LIN {X 0,Y 239.846,Z 548.939,A -85,B 0,C 180,E1 -19168.321,E2 -19168.321} C_VEL
LIN {X 0,Y 239.916,Z 549.699,A -85,B 0,C 180,E1 -19170,E2 -19170} C_VEL
LIN {X 0,Y 239.751,Z 550.198,A -85,B 0,C 180,E1 -19173.361,E2 -19173.361} C_VEL
LIN {X 0,Y 239.899,Z 549.378,A -85,B 0,C 180,E1 -19176.729,E2 -19176.729} C_VEL
LIN {X 0,Y 240.489,Z 547.237,A -85,B 0,C 180,E1 -19180.098,E2 -19180.098} C_VEL
LIN {X 0,Y 241.611,Z 543.73,A -85,B 0,C 180,E1 -19183.456,E2 -19183.456} C_VEL
LIN {X 0,Y 243.585,Z 538.761,A -85,B 0,C 180,E1 -19186.769,E2 -19186.769} C_VEL
LIN {X 0,Y 245.464,Z 533.916,A -85,B 0,C 180,E1 -19189.262,E2 -19189.262} C_VEL
LIN {X 0,Y 248.227,Z 527.144,A -85,B 0,C 180,E1 -19192.033,E2 -19192.033} C_VEL
LIN {X 0,Y 251.636,Z 518.678,A -85,B 0,C 180,E1 -19194.767,E2 -19194.767} C_VEL
LIN {X 0,Y 255.078,Z 509.872,A -85,B 0,C 180,E1 -19197.039,E2 -19197.039} C_VEL
LIN {X 0,Y 258.85,Z 499.246,A -85,B 0,C 180,E1 -19199.255,E2 -19199.255} C_VEL
LIN {X 0,Y 262.242,Z 488.539,A -85,B 0,C 180,E1 -19201.056,E2 -19201.056} C_VEL
LIN {X 0,Y 265.684,Z 476.851,A -85,B 0,C 180,E1 -19202.612,E2 -19202.612} C_VEL
LIN {X 0,Y 268.817,Z 464.011,A -85,B 0,C 180,E1 -19203.974,E2 -19203.974} C_VEL
LIN {X 0,Y 271.609,Z 450.631,A -85,B 0,C 180,E1 -19205.036,E2 -19205.036} C_VEL
LIN {X 0,Y 273.793,Z 436.72,A -85,B 0,C 180,E1 -19205.842,E2 -19205.842} C_VEL
LIN {X 0,Y 275.284,Z 422.47,A -85,B 0,C 180,E1 -19206.395,E2 -19206.395} C_VEL
LIN {X 0,Y 279.07,Z 347.973,A -85,B 0,C 180,E1 -19208.307,E2 -19208.307} C_VEL
LIN {X 0,Y 278.474,Z 345.19,A -85,B 0,C 180,E1 -19208.52,E2 -19208.52} C_VEL
LIN {X 0,Y 272.199,Z 331.36,A -85,B 0,C 180,E1 -19210.309,E2 -19210.309} C_VEL
LIN {X 0,Y 266.418,Z 320.049,A -85,B 0,C 180,E1 -19212.032,E2 -19212.032} C_VEL
LIN {X 0,Y 260.658,Z 310.039,A -85,B 0,C 180,E1 -19213.842,E2 -19213.842} C_VEL
LIN {X 0,Y 255.666,Z 301.72,A -85,B 0,C 180,E1 -19215.523,E2 -19215.523} C_VEL
LIN {X 0,Y 251.265,Z 295.251,A -85,B 0,C 180,E1 -19217.083,E2 -19217.083} C_VEL
LIN {X 0,Y 247.968,Z 290.346,A -85,B 0,C 180,E1 -19218.331,E2 -19218.331} C_VEL
LIN {X 0,Y 244.184,Z 284.789,A -85,B 0,C 180,E1 -19219.908,E2 -19219.908} C_VEL
LIN {X 0,Y 242.91,Z 280.592,A -85,B 0,C 180,E1 -19222.583,E2 -19222.583} C_VEL
LIN {X 0,Y 241.985,Z 277.932,A -85,B 0,C 180,E1 -19224.487,E2 -19224.487} C_VEL
LIN {X 0,Y 241.974,Z 277.96,A -85,B 0,C 180,E1 -19228.478,E2 -19228.478} C_VEL
LIN {X 0,Y 242.007,Z 277.954,A -85,B 0,C 180,E1 -19232.31,E2 -19232.31} C_VEL
LIN {X 0,Y 242.055,Z 277.948,A -85,B 0,C 180,E1 -19236.014,E2 -19236.014} C_VEL
LIN {X 0,Y 242.035,Z 277.95,A -85,B 0,C 180,E1 -19239.606,E2 -19239.606} C_VEL
LIN {X 0,Y 242.161,Z 277.935,A -85,B 0,C 180,E1 -19243.276,E2 -19243.276} C_VEL
LIN {X 0,Y 242.182,Z 277.929,A -85,B 0,C 180,E1 -19248.277,E2 -19248.277} C_VEL
LIN {X 0,Y 242.422,Z 277.903,A -85,B 0,C 180,E1 -19251.663,E2 -19251.663} C_VEL
LIN {X 0,Y 242.254,Z 277.935,A -85,B 0,C 180,E1 -19255.005,E2 -19255.005} C_VEL
LIN {X 0,Y 242.631,Z 277.881,A -85,B 0,C 180,E1 -19258.338,E2 -19258.338} C_VEL
LIN {X 0,Y 242.631,Z 277.874,A -85,B 0,C 180,E1 -19261.658,E2 -19261.658} C_VEL
LIN {X 0,Y 242.419,Z 277.905,A -85,B 0,C 180,E1 -19266.732,E2 -19266.732} C_VEL
LIN {X 0,Y 242.307,Z 277.915,A -85,B 0,C 180,E1 -19270.02,E2 -19270.02} C_VEL
LIN {X 0,Y 242.158,Z 277.944,A -85,B 0,C 180,E1 -19275.139,E2 -19275.139} C_VEL
LIN {X 0,Y 242.065,Z 277.955,A -85,B 0,C 180,E1 -19278.622,E2 -19278.622} C_VEL
LIN {X 0,Y 242.004,Z 277.965,A -85,B 0,C 180,E1 -19282.178,E2 -19282.178} C_VEL
LIN {X 0,Y 242.085,Z 277.957,A -85,B 0,C 180,E1 -19285.468,E2 -19285.468} C_VEL
LIN {X 0,Y 242.865,Z 280.47,A -85,B 0,C 180,E1 -19285.896,E2 -19285.896} C_VEL
LIN {X 0,Y 244.734,Z 282.697,A -85,B 0,C 180,E1 -19286.658,E2 -19286.658} C_VEL
LIN {X 0,Y 246.03,Z 283.589,A -85,B 0,C 180,E1 -19287.137,E2 -19287.137} C_VEL
LIN {X 0,Y 247.872,Z 286.714,A -85,B 0,C 180,E1 -19287.891,E2 -19287.891} C_VEL
LIN {X 0,Y 249.981,Z 289.004,A -85,B 0,C 180,E1 -19288.662,E2 -19288.662} C_VEL
LIN {X 0,Y 252.783,Z 292.768,A -85,B 0,C 180,E1 -19289.68,E2 -19289.68} C_VEL
LIN {X 0,Y 257.721,Z 299.629,A -85,B 0,C 180,E1 -19291.374,E2 -19291.374} C_VEL
LIN {X 0,Y 265.051,Z 311.16,A -85,B 0,C 180,E1 -19293.719,E2 -19293.719} C_VEL
LIN {X 0,Y 272.108,Z 323.656,A -85,B 0,C 180,E1 -19295.812,E2 -19295.812} C_VEL
LIN {X 0,Y 278.325,Z 336.16,A -85,B 0,C 180,E1 -19297.559,E2 -19297.559} C_VEL
LIN {X 0,Y 279.569,Z 338.86,A -85,B 0,C 180,E1 -19297.9,E2 -19297.9} C_VEL
LIN {X 0,Y 275.587,Z 413.281,A -85,B 0,C 180,E1 -19299.801,E2 -19299.801} C_VEL
LIN {X 0,Y 274.052,Z 427.455,A -85,B 0,C 180,E1 -19300.42,E2 -19300.42} C_VEL
LIN {X 0,Y 271.873,Z 441.305,A -85,B 0,C 180,E1 -19301.301,E2 -19301.301} C_VEL
LIN {X 0,Y 269.63,Z 452.971,A -85,B 0,C 180,E1 -19302.304,E2 -19302.304} C_VEL
LIN {X 0,Y 266.75,Z 465.144,A -85,B 0,C 180,E1 -19303.631,E2 -19303.631} C_VEL
LIN {X 0,Y 263.406,Z 477.1,A -85,B 0,C 180,E1 -19305.276,E2 -19305.276} C_VEL
LIN {X 0,Y 259.874,Z 488.093,A -85,B 0,C 180,E1 -19307.164,E2 -19307.164} C_VEL
LIN {X 0,Y 256.22,Z 498.314,A -85,B 0,C 180,E1 -19309.35,E2 -19309.35} C_VEL
LIN {X 0,Y 252.677,Z 507.464,A -85,B 0,C 180,E1 -19311.795,E2 -19311.795} C_VEL
LIN {X 0,Y 249.407,Z 515.53,A -85,B 0,C 180,E1 -19314.512,E2 -19314.512} C_VEL
LIN {X 0,Y 246.666,Z 521.907,A -85,B 0,C 180,E1 -19317.226,E2 -19317.226} C_VEL
LIN {X 0,Y 244.406,Z 527.11,A -85,B 0,C 180,E1 -19320.06,E2 -19320.06} C_VEL
LIN {X 0,Y 242.442,Z 531.556,A -85,B 0,C 180,E1 -19323.301,E2 -19323.301} C_VEL
LIN {X 0,Y 241.219,Z 534.09,A -85,B 0,C 180,E1 -19325.928,E2 -19325.928} C_VEL
LIN {X 0,Y 240.214,Z 536.197,A -85,B 0,C 180,E1 -19329.447,E2 -19329.447} C_VEL
LIN {X 0,Y 239.65,Z 536.862,A -85,B 0,C 180,E1 -19332.947,E2 -19332.947} C_VEL
LIN {X 0,Y 239.567,Z 536.099,A -85,B 0,C 180,E1 -19336.427,E2 -19336.427} C_VEL
LIN {X 0,Y 239.643,Z 533.956,A -85,B 0,C 180,E1 -19339.866,E2 -19339.866} C_VEL
LIN {X 0,Y 240.177,Z 530.391,A -85,B 0,C 180,E1 -19343.279,E2 -19343.279} C_VEL
LIN {X 0,Y 240.703,Z 526.769,A -85,B 0,C 180,E1 -19345.814,E2 -19345.814} C_VEL
LIN {X 0,Y 241.452,Z 522.2,A -85,B 0,C 180,E1 -19348.332,E2 -19348.332} C_VEL
LIN {X 0,Y 242.697,Z 515.61,A -85,B 0,C 180,E1 -19351.245,E2 -19351.245} C_VEL
LIN {X 0,Y 244.491,Z 507.418,A -85,B 0,C 180,E1 -19354.121,E2 -19354.121} C_VEL
LIN {X 0,Y 246.418,Z 498.852,A -85,B 0,C 180,E1 -19356.551,E2 -19356.551} C_VEL
LIN {X 0,Y 248.723,Z 488.467,A -85,B 0,C 180,E1 -19358.941,E2 -19358.941} C_VEL
LIN {X 0,Y 251.085,Z 477.181,A -85,B 0,C 180,E1 -19361.039,E2 -19361.039} C_VEL
LIN {X 0,Y 253.256,Z 465.291,A -85,B 0,C 180,E1 -19362.827,E2 -19362.827} C_VEL
LIN {X 0,Y 254.994,Z 454.356,A -85,B 0,C 180,E1 -19364.158,E2 -19364.158} C_VEL
LIN {X 0,Y 256.893,Z 440.565,A -85,B 0,C 180,E1 -19365.47,E2 -19365.47} C_VEL
LIN {X 0,Y 258.331,Z 426.742,A -85,B 0,C 180,E1 -19366.446,E2 -19366.446} C_VEL
LIN {X 0,Y 259.427,Z 412.336,A -85,B 0,C 180,E1 -19367.134,E2 -19367.134} C_VEL
LIN {X 0,Y 262.832,Z 324.192,A -85,B 0,C 180,E1 -19369.505,E2 -19369.505} C_VEL
LIN {X 0,Y 255.522,Z 305.251,A -85,B 0,C 180,E1 -19371.012,E2 -19371.012} C_VEL
LIN {X 0,Y 250.035,Z 293.105,A -85,B 0,C 180,E1 -19372.147,E2 -19372.147} C_VEL
LIN {X 0,Y 242.324,Z 279.276,A -85,B 0,C 180,E1 -19373.732,E2 -19373.732} C_VEL
LIN {X 0,Y 242.049,Z 277.961,A -85,B 0,C 180,E1 -19373.835,E2 -19373.835} C_VEL
LIN {X 0,Y 241.998,Z 277.966,A -85,B 0,C 180,E1 -19377.688,E2 -19377.688} C_VEL
LIN {X 0,Y 241.965,Z 277.968,A -85,B 0,C 180,E1 -19381.521,E2 -19381.521} C_VEL
LIN {X 0,Y 242.018,Z 277.961,A -85,B 0,C 180,E1 -19385.605,E2 -19385.605} C_VEL
LIN {X 0,Y 241.999,Z 277.956,A -85,B 0,C 180,E1 -19389.71,E2 -19389.71} C_VEL
LIN {X 0,Y 242,Z 277.963,A -85,B 0,C 180,E1 -19394.185,E2 -19394.185} C_VEL
LIN {X 0,Y 242.027,Z 277.954,A -85,B 0,C 180,E1 -19398.1,E2 -19398.1} C_VEL
LIN {X 0,Y 242.003,Z 277.958,A -85,B 0,C 180,E1 -19402.424,E2 -19402.424} C_VEL
LIN {X 0,Y 241.982,Z 277.959,A -85,B 0,C 180,E1 -19406.511,E2 -19406.511} C_VEL
LIN {X 0,Y 242.028,Z 277.956,A -85,B 0,C 180,E1 -19410.589,E2 -19410.589} C_VEL
LIN {X 0,Y 242.06,Z 277.941,A -85,B 0,C 180,E1 -19414.185,E2 -19414.185} C_VEL
LIN {X 0,Y 242.046,Z 277.959,A -85,B 0,C 180,E1 -19418.299,E2 -19418.299} C_VEL
LIN {X 0,Y 242.157,Z 277.945,A -85,B 0,C 180,E1 -19423.28,E2 -19423.28} C_VEL
LIN {X 0,Y 242.174,Z 277.943,A -85,B 0,C 180,E1 -19428.282,E2 -19428.282} C_VEL
LIN {X 0,Y 242.395,Z 277.902,A -85,B 0,C 180,E1 -19431.667,E2 -19431.667} C_VEL
LIN {X 0,Y 242.253,Z 277.923,A -85,B 0,C 180,E1 -19435.009,E2 -19435.009} C_VEL
LIN {X 0,Y 242.632,Z 277.888,A -85,B 0,C 180,E1 -19438.342,E2 -19438.342} C_VEL
LIN {X 0,Y 242.632,Z 277.873,A -85,B 0,C 180,E1 -19441.662,E2 -19441.662} C_VEL
LIN {X 0,Y 242.365,Z 277.899,A -85,B 0,C 180,E1 -19443.351,E2 -19443.351} C_VEL
LIN {X 0,Y 241.593,Z 278.005,A -85,B 0,C 180,E1 -19444.738,E2 -19444.738} C_VEL
LIN {X 0,Y 238.745,Z 278.37,A -85,B 0,C 180,E1 -19447.002,E2 -19447.002} C_VEL
LIN {X 0,Y 235.536,Z 278.767,A -85,B 0,C 180,E1 -19449.792,E2 -19449.792} C_VEL
LIN {X 0,Y 235.167,Z 278.802,A -85,B 0,C 180,E1 -19450.758,E2 -19450.758} C_VEL
LIN {X 0,Y 235.105,Z 278.82,A -85,B 0,C 180,E1 -19455.609,E2 -19455.609} C_VEL
LIN {X 0,Y 235.005,Z 278.83,A -85,B 0,C 180,E1 -19459.208,E2 -19459.208} C_VEL
LIN {X 0,Y 234.952,Z 278.839,A -85,B 0,C 180,E1 -19462.886,E2 -19462.886} C_VEL
LIN {X 0,Y 234.97,Z 278.838,A -85,B 0,C 180,E1 -19466.659,E2 -19466.659} C_VEL
LIN {X 0,Y 234.933,Z 278.842,A -85,B 0,C 180,E1 -19470.57,E2 -19470.57} C_VEL
LIN {X 0,Y 234.935,Z 278.843,A -85,B 0,C 180,E1 -19474.639,E2 -19474.639} C_VEL
LIN {X 0,Y 234.944,Z 278.845,A -85,B 0,C 180,E1 -19478.946,E2 -19478.946} C_VEL
LIN {X 0,Y 234.89,Z 278.85,A -85,B 0,C 180,E1 -19483.488,E2 -19483.488} C_VEL
LIN {X 0,Y 234.895,Z 278.874,A -85,B 0,C 180,E1 -19488.167,E2 -19488.167} C_VEL
LIN {X 0,Y 236.892,Z 286.452,A -85,B 0,C 180,E1 -19491.308,E2 -19491.308} C_VEL
LIN {X 0,Y 244.745,Z 303.391,A -85,B 0,C 180,E1 -19493.084,E2 -19493.084} C_VEL
LIN {X 0,Y 252.555,Z 322.958,A -85,B 0,C 180,E1 -19494.805,E2 -19494.805} C_VEL
LIN {X 0,Y 253.857,Z 327.02,A -85,B 0,C 180,E1 -19495.104,E2 -19495.104} C_VEL
LIN {X 0,Y 256.076,Z 343.908,A -85,B 0,C 180,E1 -19495.922,E2 -19495.922} C_VEL
LIN {X 0,Y 252.934,Z 424.435,A -85,B 0,C 180,E1 -19498.135,E2 -19498.135} C_VEL
LIN {X 0,Y 251.91,Z 437.762,A -85,B 0,C 180,E1 -19498.752,E2 -19498.752} C_VEL
LIN {X 0,Y 250.233,Z 451.111,A -85,B 0,C 180,E1 -19499.633,E2 -19499.633} C_VEL
LIN {X 0,Y 248.32,Z 463.814,A -85,B 0,C 180,E1 -19500.777,E2 -19500.777} C_VEL
LIN {X 0,Y 246.163,Z 476.754,A -85,B 0,C 180,E1 -19502.311,E2 -19502.311} C_VEL
LIN {X 0,Y 244.22,Z 486.606,A -85,B 0,C 180,E1 -19503.74,E2 -19503.74} C_VEL
LIN {X 0,Y 241.878,Z 497.961,A -85,B 0,C 180,E1 -19505.769,E2 -19505.769} C_VEL
LIN {X 0,Y 239.496,Z 508.241,A -85,B 0,C 180,E1 -19508.029,E2 -19508.029} C_VEL
LIN {X 0,Y 237.408,Z 517.546,A -85,B 0,C 180,E1 -19510.547,E2 -19510.547} C_VEL
LIN {X 0,Y 235.808,Z 525.288,A -85,B 0,C 180,E1 -19513.107,E2 -19513.107} C_VEL
LIN {X 0,Y 234.372,Z 532.651,A -85,B 0,C 180,E1 -19516.12,E2 -19516.12} C_VEL
LIN {X 0,Y 233.48,Z 537.791,A -85,B 0,C 180,E1 -19518.717,E2 -19518.717} C_VEL
LIN {X 0,Y 232.927,Z 543.07,A -85,B 0,C 180,E1 -19522.196,E2 -19522.196} C_VEL
LIN {X 0,Y 232.701,Z 546.505,A -85,B 0,C 180,E1 -19525.335,E2 -19525.335} C_VEL
LIN {X 0,Y 232.758,Z 548.66,A -85,B 0,C 180,E1 -19528.27,E2 -19528.27} C_VEL
LIN {X 0,Y 232.825,Z 549.454,A -85,B 0,C 180,E1 -19530,E2 -19530} C_VEL
LIN {X 0,Y 232.662,Z 550.012,A -85,B 0,C 180,E1 -19533.463,E2 -19533.463} C_VEL
LIN {X 0,Y 232.82,Z 549.246,A -85,B 0,C 180,E1 -19536.935,E2 -19536.935} C_VEL
LIN {X 0,Y 233.47,Z 547.162,A -85,B 0,C 180,E1 -19540.405,E2 -19540.405} C_VEL
LIN {X 0,Y 234.687,Z 543.715,A -85,B 0,C 180,E1 -19543.861,E2 -19543.861} C_VEL
LIN {X 0,Y 236.758,Z 538.813,A -85,B 0,C 180,E1 -19547.267,E2 -19547.267} C_VEL
LIN {X 0,Y 238.627,Z 534.303,A -85,B 0,C 180,E1 -19549.707,E2 -19549.707} C_VEL
LIN {X 0,Y 241.645,Z 527.347,A -85,B 0,C 180,E1 -19552.666,E2 -19552.666} C_VEL
LIN {X 0,Y 245.222,Z 518.966,A -85,B 0,C 180,E1 -19555.46,E2 -19555.46} C_VEL
LIN {X 0,Y 248.79,Z 510.258,A -85,B 0,C 180,E1 -19557.781,E2 -19557.781} C_VEL
LIN {X 0,Y 252.717,Z 499.747,A -85,B 0,C 180,E1 -19560.037,E2 -19560.037} C_VEL
LIN {X 0,Y 256.218,Z 489.183,A -85,B 0,C 180,E1 -19561.871,E2 -19561.871} C_VEL
LIN {X 0,Y 259.781,Z 477.673,A -85,B 0,C 180,E1 -19563.449,E2 -19563.449} C_VEL
LIN {X 0,Y 263.013,Z 465.076,A -85,B 0,C 180,E1 -19564.83,E2 -19564.83} C_VEL
LIN {X 0,Y 265.898,Z 452.049,A -85,B 0,C 180,E1 -19565.904,E2 -19565.904} C_VEL
LIN {X 0,Y 268.244,Z 438.06,A -85,B 0,C 180,E1 -19566.762,E2 -19566.762} C_VEL
LIN {X 0,Y 269.928,Z 423.494,A -85,B 0,C 180,E1 -19567.36,E2 -19567.36} C_VEL
LIN {X 0,Y 273.887,Z 349.141,A -85,B 0,C 180,E1 -19569.299,E2 -19569.299} C_VEL
LIN {X 0,Y 268.082,Z 336.015,A -85,B 0,C 180,E1 -19571.032,E2 -19571.032} C_VEL
LIN {X 0,Y 262.07,Z 324.165,A -85,B 0,C 180,E1 -19572.906,E2 -19572.906} C_VEL
LIN {X 0,Y 256.592,Z 314.442,A -85,B 0,C 180,E1 -19574.715,E2 -19574.715} C_VEL
LIN {X 0,Y 251.898,Z 306.619,A -85,B 0,C 180,E1 -19576.369,E2 -19576.369} C_VEL
LIN {X 0,Y 248.032,Z 300.769,A -85,B 0,C 180,E1 -19577.805,E2 -19577.805} C_VEL
LIN {X 0,Y 244.753,Z 295.838,A -85,B 0,C 180,E1 -19579.097,E2 -19579.097} C_VEL
LIN {X 0,Y 240.658,Z 290.029,A -85,B 0,C 180,E1 -19580.81,E2 -19580.81} C_VEL
LIN {X 0,Y 237.369,Z 285.469,A -85,B 0,C 180,E1 -19582.294,E2 -19582.294} C_VEL
LIN {X 0,Y 236.895,Z 284.516,A -85,B 0,C 180,E1 -19582.541,E2 -19582.541} C_VEL
LIN {X 0,Y 235.976,Z 281.719,A -85,B 0,C 180,E1 -19584.526,E2 -19584.526} C_VEL
LIN {X 0,Y 234.943,Z 278.838,A -85,B 0,C 180,E1 -19586.883,E2 -19586.883} C_VEL
LIN {X 0,Y 234.951,Z 278.837,A -85,B 0,C 180,E1 -19591.404,E2 -19591.404} C_VEL
LIN {X 0,Y 234.986,Z 278.831,A -85,B 0,C 180,E1 -19595.244,E2 -19595.244} C_VEL
LIN {X 0,Y 235.009,Z 278.829,A -85,B 0,C 180,E1 -19598.967,E2 -19598.967} C_VEL
LIN {X 0,Y 235.094,Z 278.817,A -85,B 0,C 180,E1 -19603.057,E2 -19603.057} C_VEL
LIN {X 0,Y 235.114,Z 278.81,A -85,B 0,C 180,E1 -19607.92,E2 -19607.92} C_VEL
LIN {X 0,Y 235.371,Z 278.783,A -85,B 0,C 180,E1 -19611.412,E2 -19611.412} C_VEL
LIN {X 0,Y 235.398,Z 278.775,A -85,B 0,C 180,E1 -19613.139,E2 -19613.139} C_VEL
LIN {X 0,Y 235.59,Z 278.757,A -85,B 0,C 180,E1 -19618.288,E2 -19618.288} C_VEL
LIN {X 0,Y 235.59,Z 278.751,A -85,B 0,C 180,E1 -19621.707,E2 -19621.707} C_VEL
LIN {X 0,Y 235.395,Z 278.782,A -85,B 0,C 180,E1 -19626.856,E2 -19626.856} C_VEL
LIN {X 0,Y 235.231,Z 278.798,A -85,B 0,C 180,E1 -19630.324,E2 -19630.324} C_VEL
LIN {X 0,Y 235.105,Z 278.825,A -85,B 0,C 180,E1 -19635.604,E2 -19635.604} C_VEL
LIN {X 0,Y 235.001,Z 278.838,A -85,B 0,C 180,E1 -19639.204,E2 -19639.204} C_VEL
LIN {X 0,Y 234.95,Z 278.859,A -85,B 0,C 180,E1 -19642.781,E2 -19642.781} C_VEL
LIN {X 0,Y 235.678,Z 281.125,A -85,B 0,C 180,E1 -19643.212,E2 -19643.212} C_VEL
LIN {X 0,Y 237.389,Z 283.308,A -85,B 0,C 180,E1 -19644.018,E2 -19644.018} C_VEL
LIN {X 0,Y 239.259,Z 284.698,A -85,B 0,C 180,E1 -19644.811,E2 -19644.811} C_VEL
LIN {X 0,Y 241.156,Z 287.891,A -85,B 0,C 180,E1 -19645.682,E2 -19645.682} C_VEL
LIN {X 0,Y 243.288,Z 289.963,A -85,B 0,C 180,E1 -19646.539,E2 -19646.539} C_VEL
LIN {X 0,Y 245.784,Z 293.515,A -85,B 0,C 180,E1 -19647.553,E2 -19647.553} C_VEL
LIN {X 0,Y 247.214,Z 295.215,A -85,B 0,C 180,E1 -19648.097,E2 -19648.097} C_VEL
LIN {X 0,Y 251.651,Z 301.325,A -85,B 0,C 180,E1 -19649.744,E2 -19649.744} C_VEL
LIN {X 0,Y 254.449,Z 305.277,A -85,B 0,C 180,E1 -19650.726,E2 -19650.726} C_VEL
LIN {X 0,Y 260.415,Z 314.765,A -85,B 0,C 180,E1 -19652.721,E2 -19652.721} C_VEL
LIN {X 0,Y 267.954,Z 328.174,A -85,B 0,C 180,E1 -19655.066,E2 -19655.066} C_VEL
LIN {X 0,Y 274.346,Z 341.366,A -85,B 0,C 180,E1 -19656.94,E2 -19656.94} C_VEL
LIN {X 0,Y 270.329,Z 413.322,A -85,B 0,C 180,E1 -19658.8,E2 -19658.8} C_VEL
LIN {X 0,Y 268.827,Z 426.929,A -85,B 0,C 180,E1 -19659.391,E2 -19659.391} C_VEL
LIN {X 0,Y 266.564,Z 440.953,A -85,B 0,C 180,E1 -19660.278,E2 -19660.278} C_VEL
LIN {X 0,Y 264.231,Z 452.729,A -85,B 0,C 180,E1 -19661.291,E2 -19661.291} C_VEL
LIN {X 0,Y 261.073,Z 465.573,A -85,B 0,C 180,E1 -19662.706,E2 -19662.706} C_VEL
LIN {X 0,Y 257.766,Z 477.003,A -85,B 0,C 180,E1 -19664.3,E2 -19664.3} C_VEL
LIN {X 0,Y 253.994,Z 488.173,A -85,B 0,C 180,E1 -19666.233,E2 -19666.233} C_VEL
LIN {X 0,Y 250.566,Z 497.454,A -85,B 0,C 180,E1 -19668.231,E2 -19668.231} C_VEL
LIN {X 0,Y 246.677,Z 507.097,A -85,B 0,C 180,E1 -19670.807,E2 -19670.807} C_VEL
LIN {X 0,Y 243.602,Z 514.299,A -85,B 0,C 180,E1 -19673.217,E2 -19673.217} C_VEL
LIN {X 0,Y 240.379,Z 521.525,A -85,B 0,C 180,E1 -19676.255,E2 -19676.255} C_VEL
LIN {X 0,Y 238.141,Z 526.34,A -85,B 0,C 180,E1 -19678.848,E2 -19678.848} C_VEL
LIN {X 0,Y 236.223,Z 530.325,A -85,B 0,C 180,E1 -19681.575,E2 -19681.575} C_VEL
LIN {X 0,Y 234.408,Z 534.057,A -85,B 0,C 180,E1 -19685.182,E2 -19685.182} C_VEL
LIN {X 0,Y 233.261,Z 536.272,A -85,B 0,C 180,E1 -19688.805,E2 -19688.805} C_VEL
LIN {X 0,Y 232.611,Z 537.05,A -85,B 0,C 180,E1 -19692.415,E2 -19692.415} C_VEL
LIN {X 0,Y 232.472,Z 536.422,A -85,B 0,C 180,E1 -19696.005,E2 -19696.005} C_VEL
LIN {X 0,Y 232.51,Z 534.393,A -85,B 0,C 180,E1 -19699.551,E2 -19699.551} C_VEL
LIN {X 0,Y 233.037,Z 530.933,A -85,B 0,C 180,E1 -19703.072,E2 -19703.072} C_VEL
LIN {X 0,Y 233.59,Z 527.399,A -85,B 0,C 180,E1 -19705.687,E2 -19705.687} C_VEL
LIN {X 0,Y 234.327,Z 522.912,A -85,B 0,C 180,E1 -19708.282,E2 -19708.282} C_VEL
LIN {X 0,Y 235.573,Z 516.449,A -85,B 0,C 180,E1 -19711.282,E2 -19711.282} C_VEL
LIN {X 0,Y 237.073,Z 509.657,A -85,B 0,C 180,E1 -19713.825,E2 -19713.825} C_VEL
LIN {X 0,Y 239.011,Z 501.501,A -85,B 0,C 180,E1 -19716.331,E2 -19716.331} C_VEL
LIN {X 0,Y 241.287,Z 491.679,A -85,B 0,C 180,E1 -19718.796,E2 -19718.796} C_VEL
LIN {X 0,Y 243.625,Z 481.194,A -85,B 0,C 180,E1 -19720.934,E2 -19720.934} C_VEL
LIN {X 0,Y 245.841,Z 469.979,A -85,B 0,C 180,E1 -19722.8,E2 -19722.8} C_VEL
LIN {X 0,Y 247.81,Z 458.365,A -85,B 0,C 180,E1 -19724.368,E2 -19724.368} C_VEL
LIN {X 0,Y 249.896,Z 445.634,A -85,B 0,C 180,E1 -19725.705,E2 -19725.705} C_VEL
LIN {X 0,Y 251.534,Z 431.462,A -85,B 0,C 180,E1 -19726.851,E2 -19726.851} C_VEL
LIN {X 0,Y 252.743,Z 417.083,A -85,B 0,C 180,E1 -19727.654,E2 -19727.654} C_VEL
LIN {X 0,Y 253.645,Z 400.006,A -85,B 0,C 180,E1 -19728.22,E2 -19728.22} C_VEL
LIN {X 0,Y 256.575,Z 325.836,A -85,B 0,C 180,E1 -19730.218,E2 -19730.218} C_VEL
LIN {X 0,Y 248.954,Z 306.387,A -85,B 0,C 180,E1 -19731.853,E2 -19731.853} C_VEL
LIN {X 0,Y 244.442,Z 296.468,A -85,B 0,C 180,E1 -19732.824,E2 -19732.824} C_VEL
LIN {X 0,Y 236.349,Z 282.205,A -85,B 0,C 180,E1 -19734.556,E2 -19734.556} C_VEL
LIN {X 0,Y 235.072,Z 279.404,A -85,B 0,C 180,E1 -19734.864,E2 -19734.864} C_VEL
LIN {X 0,Y 234.99,Z 278.833,A -85,B 0,C 180,E1 -19734.933,E2 -19734.933} C_VEL
LIN {X 0,Y 234.958,Z 278.832,A -85,B 0,C 180,E1 -19739.844,E2 -19739.844} C_VEL
LIN {X 0,Y 234.95,Z 278.843,A -85,B 0,C 180,E1 -19744.634,E2 -19744.634} C_VEL
LIN {X 0,Y 234.957,Z 278.84,A -85,B 0,C 180,E1 -19748.953,E2 -19748.953} C_VEL
LIN {X 0,Y 234.983,Z 278.84,A -85,B 0,C 180,E1 -19753.463,E2 -19753.463} C_VEL
LIN {X 0,Y 234.986,Z 278.824,A -85,B 0,C 180,E1 -19756.541,E2 -19756.541} C_VEL
LIN {X 0,Y 234.946,Z 278.842,A -85,B 0,C 180,E1 -19761.088,E2 -19761.088} C_VEL
LIN {X 0,Y 234.952,Z 278.827,A -85,B 0,C 180,E1 -19765.369,E2 -19765.369} C_VEL
LIN {X 0,Y 234.961,Z 278.837,A -85,B 0,C 180,E1 -19770.159,E2 -19770.159} C_VEL
LIN {X 0,Y 234.987,Z 278.819,A -85,B 0,C 180,E1 -19773.796,E2 -19773.796} C_VEL
LIN {X 0,Y 235.004,Z 278.835,A -85,B 0,C 180,E1 -19778.972,E2 -19778.972} C_VEL
LIN {X 0,Y 235.09,Z 278.826,A -85,B 0,C 180,E1 -19783.062,E2 -19783.062} C_VEL
LIN {X 0,Y 235.108,Z 278.822,A -85,B 0,C 180,E1 -19787.924,E2 -19787.924} C_VEL
LIN {X 0,Y 235.326,Z 278.782,A -85,B 0,C 180,E1 -19791.415,E2 -19791.415} C_VEL
LIN {X 0,Y 235.368,Z 278.768,A -85,B 0,C 180,E1 -19793.143,E2 -19793.143} C_VEL
LIN {X 0,Y 235.591,Z 278.764,A -85,B 0,C 180,E1 -19798.293,E2 -19798.293} C_VEL
LIN {X 0,Y 235.591,Z 278.748,A -85,B 0,C 180,E1 -19801.712,E2 -19801.712} C_VEL
LIN {X 0,Y 235.37,Z 278.791,A -85,B 0,C 180,E1 -19806.862,E2 -19806.862} C_VEL
LIN {X 0,Y 235.167,Z 278.802,A -85,B 0,C 180,E1 -19810.758,E2 -19810.758} C_VEL
LIN {X 0,Y 234.424,Z 278.89,A -85,B 0,C 180,E1 -19812.186,E2 -19812.186} C_VEL
LIN {X 0,Y 231.562,Z 279.256,A -85,B 0,C 180,E1 -19814.517,E2 -19814.517} C_VEL
LIN {X 0,Y 228.324,Z 279.67,A -85,B 0,C 180,E1 -19817.393,E2 -19817.393} C_VEL
LIN {X 0,Y 227.964,Z 279.71,A -85,B 0,C 180,E1 -19818.389,E2 -19818.389} C_VEL
LIN {X 0,Y 227.916,Z 279.718,A -85,B 0,C 180,E1 -19822.323,E2 -19822.323} C_VEL
LIN {X 0,Y 227.943,Z 279.713,A -85,B 0,C 180,E1 -19826.605,E2 -19826.605} C_VEL
LIN {X 0,Y 227.91,Z 279.718,A -85,B 0,C 180,E1 -19830.298,E2 -19830.298} C_VEL
LIN {X 0,Y 227.88,Z 279.724,A -85,B 0,C 180,E1 -19833.722,E2 -19833.722} C_VEL
LIN {X 0,Y 227.848,Z 279.728,A -85,B 0,C 180,E1 -19838.093,E2 -19838.093} C_VEL
LIN {X 0,Y 227.813,Z 279.73,A -85,B 0,C 180,E1 -19842.744,E2 -19842.744} C_VEL
LIN {X 0,Y 227.871,Z 279.875,A -85,B 0,C 180,E1 -19847.349,E2 -19847.349} C_VEL
LIN {X 0,Y 229.601,Z 286.436,A -85,B 0,C 180,E1 -19850.115,E2 -19850.115} C_VEL
LIN {X 0,Y 237.198,Z 302.109,A -85,B 0,C 180,E1 -19851.915,E2 -19851.915} C_VEL
LIN {X 0,Y 245.113,Z 321.434,A -85,B 0,C 180,E1 -19853.75,E2 -19853.75} C_VEL
LIN {X 0,Y 247.823,Z 329.009,A -85,B 0,C 180,E1 -19854.376,E2 -19854.376} C_VEL
LIN {X 0,Y 249.832,Z 344.992,A -85,B 0,C 180,E1 -19855.17,E2 -19855.17} C_VEL
LIN {X 0,Y 246.618,Z 424.352,A -85,B 0,C 180,E1 -19857.4,E2 -19857.4} C_VEL
LIN {X 0,Y 245.553,Z 437.636,A -85,B 0,C 180,E1 -19858.03,E2 -19858.03} C_VEL
LIN {X 0,Y 243.742,Z 451.535,A -85,B 0,C 180,E1 -19858.976,E2 -19858.976} C_VEL
LIN {X 0,Y 241.771,Z 464.106,A -85,B 0,C 180,E1 -19860.146,E2 -19860.146} C_VEL
LIN {X 0,Y 239.692,Z 476.142,A -85,B 0,C 180,E1 -19861.601,E2 -19861.601} C_VEL
LIN {X 0,Y 237.541,Z 486.761,A -85,B 0,C 180,E1 -19863.18,E2 -19863.18} C_VEL
LIN {X 0,Y 235.103,Z 498.043,A -85,B 0,C 180,E1 -19865.26,E2 -19865.26} C_VEL
LIN {X 0,Y 232.864,Z 507.452,A -85,B 0,C 180,E1 -19867.369,E2 -19867.369} C_VEL
LIN {X 0,Y 230.654,Z 516.861,A -85,B 0,C 180,E1 -19869.954,E2 -19869.954} C_VEL
LIN {X 0,Y 228.88,Z 524.684,A -85,B 0,C 180,E1 -19872.58,E2 -19872.58} C_VEL
LIN {X 0,Y 227.425,Z 532.131,A -85,B 0,C 180,E1 -19875.687,E2 -19875.687} C_VEL
LIN {X 0,Y 226.476,Z 537.32,A -85,B 0,C 180,E1 -19878.363,E2 -19878.363} C_VEL
LIN {X 0,Y 225.971,Z 541.477,A -85,B 0,C 180,E1 -19881.054,E2 -19881.054} C_VEL
LIN {X 0,Y 225.648,Z 545.659,A -85,B 0,C 180,E1 -19884.639,E2 -19884.639} C_VEL
LIN {X 0,Y 225.672,Z 548.366,A -85,B 0,C 180,E1 -19888.215,E2 -19888.215} C_VEL
LIN {X 0,Y 225.737,Z 549.194,A -85,B 0,C 180,E1 -19890,E2 -19890} C_VEL
LIN {X 0,Y 225.577,Z 549.817,A -85,B 0,C 180,E1 -19893.572,E2 -19893.572} C_VEL
LIN {X 0,Y 225.767,Z 549.114,A -85,B 0,C 180,E1 -19897.153,E2 -19897.153} C_VEL
LIN {X 0,Y 226.465,Z 547.091,A -85,B 0,C 180,E1 -19900.731,E2 -19900.731} C_VEL
LIN {X 0,Y 227.781,Z 543.707,A -85,B 0,C 180,E1 -19904.29,E2 -19904.29} C_VEL
LIN {X 0,Y 229.955,Z 538.87,A -85,B 0,C 180,E1 -19907.795,E2 -19907.795} C_VEL
LIN {X 0,Y 231.935,Z 534.413,A -85,B 0,C 180,E1 -19910.3,E2 -19910.3} C_VEL
LIN {X 0,Y 235.11,Z 527.548,A -85,B 0,C 180,E1 -19913.332,E2 -19913.332} C_VEL
LIN {X 0,Y 238.823,Z 519.255,A -85,B 0,C 180,E1 -19916.193,E2 -19916.193} C_VEL
LIN {X 0,Y 242.551,Z 510.644,A -85,B 0,C 180,E1 -19918.56,E2 -19918.56} C_VEL
LIN {X 0,Y 246.633,Z 500.254,A -85,B 0,C 180,E1 -19920.858,E2 -19920.858} C_VEL
LIN {X 0,Y 250.251,Z 489.843,A -85,B 0,C 180,E1 -19922.724,E2 -19922.724} C_VEL
LIN {X 0,Y 253.929,Z 478.525,A -85,B 0,C 180,E1 -19924.326,E2 -19924.326} C_VEL
LIN {X 0,Y 257.272,Z 466.189,A -85,B 0,C 180,E1 -19925.725,E2 -19925.725} C_VEL
LIN {X 0,Y 260.473,Z 452.415,A -85,B 0,C 180,E1 -19926.893,E2 -19926.893} C_VEL
LIN {X 0,Y 262.886,Z 438.624,A -85,B 0,C 180,E1 -19927.76,E2 -19927.76} C_VEL
LIN {X 0,Y 264.654,Z 424.227,A -85,B 0,C 180,E1 -19928.373,E2 -19928.373} C_VEL
LIN {X 0,Y 268.796,Z 352.724,A -85,B 0,C 180,E1 -19930.238,E2 -19930.238} C_VEL
LIN {X 0,Y 268.574,Z 351.171,A -85,B 0,C 180,E1 -19930.345,E2 -19930.345} C_VEL
LIN {X 0,Y 262.793,Z 338.113,A -85,B 0,C 180,E1 -19932.165,E2 -19932.165} C_VEL
LIN {X 0,Y 256.32,Z 325.359,A -85,B 0,C 180,E1 -19934.317,E2 -19934.317} C_VEL
LIN {X 0,Y 248.927,Z 312.488,A -85,B 0,C 180,E1 -19936.973,E2 -19936.973} C_VEL
LIN {X 0,Y 244.705,Z 306.031,A -85,B 0,C 180,E1 -19938.603,E2 -19938.603} C_VEL
LIN {X 0,Y 241.619,Z 301.345,A -85,B 0,C 180,E1 -19939.872,E2 -19939.872} C_VEL
LIN {X 0,Y 237.823,Z 295.786,A -85,B 0,C 180,E1 -19941.541,E2 -19941.541} C_VEL
LIN {X 0,Y 234.471,Z 290.981,A -85,B 0,C 180,E1 -19943.125,E2 -19943.125} C_VEL
LIN {X 0,Y 229.481,Z 284.428,A -85,B 0,C 180,E1 -19945.684,E2 -19945.684} C_VEL
LIN {X 0,Y 229.058,Z 283.21,A -85,B 0,C 180,E1 -19946.474,E2 -19946.474} C_VEL
LIN {X 0,Y 227.892,Z 279.714,A -85,B 0,C 180,E1 -19949.497,E2 -19949.497} C_VEL
LIN {X 0,Y 227.928,Z 279.719,A -85,B 0,C 180,E1 -19954.423,E2 -19954.423} C_VEL
LIN {X 0,Y 227.96,Z 279.714,A -85,B 0,C 180,E1 -19958.285,E2 -19958.285} C_VEL
LIN {X 0,Y 228.032,Z 279.698,A -85,B 0,C 180,E1 -19962.824,E2 -19962.824} C_VEL
LIN {X 0,Y 228.071,Z 279.689,A -85,B 0,C 180,E1 -19967.541,E2 -19967.541} C_VEL
LIN {X 0,Y 228.301,Z 279.667,A -85,B 0,C 180,E1 -19971.144,E2 -19971.144} C_VEL
LIN {X 0,Y 228.349,Z 279.652,A -85,B 0,C 180,E1 -19972.926,E2 -19972.926} C_VEL
LIN {X 0,Y 228.549,Z 279.633,A -85,B 0,C 180,E1 -19978.236,E2 -19978.236} C_VEL
LIN {X 0,Y 228.549,Z 279.628,A -85,B 0,C 180,E1 -19981.76,E2 -19981.76} C_VEL
LIN {X 0,Y 228.347,Z 279.662,A -85,B 0,C 180,E1 -19987.069,E2 -19987.069} C_VEL
LIN {X 0,Y 228.156,Z 279.681,A -85,B 0,C 180,E1 -19990.648,E2 -19990.648} C_VEL
LIN {X 0,Y 228.056,Z 279.692,A -85,B 0,C 180,E1 -19994.27,E2 -19994.27} C_VEL
LIN {X 0,Y 227.995,Z 279.701,A -85,B 0,C 180,E1 -19997.951,E2 -19997.951} C_VEL
LIN {X 0,Y 227.941,Z 279.755,A -85,B 0,C 180,E1 -19999.705,E2 -19999.705} C_VEL
LIN {X 0,Y 228.778,Z 282.281,A -85,B 0,C 180,E1 -20000.274,E2 -20000.274} C_VEL
LIN {X 0,Y 230.738,Z 284.516,A -85,B 0,C 180,E1 -20001.319,E2 -20001.319} C_VEL
LIN {X 0,Y 232.4,Z 285.686,A -85,B 0,C 180,E1 -20002.12,E2 -20002.12} C_VEL
LIN {X 0,Y 234.227,Z 288.769,A -85,B 0,C 180,E1 -20003.073,E2 -20003.073} C_VEL
LIN {X 0,Y 236.725,Z 291.144,A -85,B 0,C 180,E1 -20004.206,E2 -20004.206} C_VEL
LIN {X 0,Y 239.079,Z 294.527,A -85,B 0,C 180,E1 -20005.285,E2 -20005.285} C_VEL
LIN {X 0,Y 240.704,Z 296.342,A -85,B 0,C 180,E1 -20005.971,E2 -20005.971} C_VEL
LIN {X 0,Y 245.046,Z 302.223,A -85,B 0,C 180,E1 -20007.747,E2 -20007.747} C_VEL
LIN {X 0,Y 248.059,Z 306.297,A -85,B 0,C 180,E1 -20008.898,E2 -20008.898} C_VEL
LIN {X 0,Y 251.32,Z 311.051,A -85,B 0,C 180,E1 -20010.096,E2 -20010.096} C_VEL
LIN {X 0,Y 257.58,Z 321.227,A -85,B 0,C 180,E1 -20012.265,E2 -20012.265} C_VEL
LIN {X 0,Y 264.848,Z 334.67,A -85,B 0,C 180,E1 -20014.61,E2 -20014.61} C_VEL
LIN {X 0,Y 269.13,Z 343.742,A -85,B 0,C 180,E1 -20015.923,E2 -20015.923} C_VEL
LIN {X 0,Y 265.17,Z 413.405,A -85,B 0,C 180,E1 -20017.76,E2 -20017.76} C_VEL
LIN {X 0,Y 263.54,Z 427.483,A -85,B 0,C 180,E1 -20018.378,E2 -20018.378} C_VEL
LIN {X 0,Y 261.341,Z 440.65,A -85,B 0,C 180,E1 -20019.213,E2 -20019.213} C_VEL
LIN {X 0,Y 258.923,Z 452.537,A -85,B 0,C 180,E1 -20020.237,E2 -20020.237} C_VEL
LIN {X 0,Y 255.588,Z 465.62,A -85,B 0,C 180,E1 -20021.688,E2 -20021.688} C_VEL
LIN {X 0,Y 251.806,Z 478.158,A -85,B 0,C 180,E1 -20023.477,E2 -20023.477} C_VEL
LIN {X 0,Y 247.886,Z 489.154,A -85,B 0,C 180,E1 -20025.438,E2 -20025.438} C_VEL
LIN {X 0,Y 244.331,Z 498.298,A -85,B 0,C 180,E1 -20027.473,E2 -20027.473} C_VEL
LIN {X 0,Y 240.472,Z 507.442,A -85,B 0,C 180,E1 -20029.988,E2 -20029.988} C_VEL
LIN {X 0,Y 237.063,Z 514.962,A -85,B 0,C 180,E1 -20032.575,E2 -20032.575} C_VEL
LIN {X 0,Y 234.125,Z 521.138,A -85,B 0,C 180,E1 -20035.227,E2 -20035.227} C_VEL
LIN {X 0,Y 231.425,Z 526.66,A -85,B 0,C 180,E1 -20038.24,E2 -20038.24} C_VEL
LIN {X 0,Y 229.078,Z 531.283,A -85,B 0,C 180,E1 -20041.607,E2 -20041.607} C_VEL
LIN {X 0,Y 227.635,Z 534.028,A -85,B 0,C 180,E1 -20044.391,E2 -20044.391} C_VEL
LIN {X 0,Y 226.328,Z 536.349,A -85,B 0,C 180,E1 -20048.123,E2 -20048.123} C_VEL
LIN {X 0,Y 225.569,Z 537.23,A -85,B 0,C 180,E1 -20051.847,E2 -20051.847} C_VEL
LIN {X 0,Y 225.372,Z 536.708,A -85,B 0,C 180,E1 -20055.554,E2 -20055.554} C_VEL
LIN {X 0,Y 225.383,Z 534.81,A -85,B 0,C 180,E1 -20059.217,E2 -20059.217} C_VEL
LIN {X 0,Y 225.889,Z 531.473,A -85,B 0,C 180,E1 -20062.851,E2 -20062.851} C_VEL
LIN {X 0,Y 226.473,Z 527.99,A -85,B 0,C 180,E1 -20065.551,E2 -20065.551} C_VEL
LIN {X 0,Y 227.523,Z 521.986,A -85,B 0,C 180,E1 -20069.115,E2 -20069.115} C_VEL
LIN {X 0,Y 228.967,Z 515.219,A -85,B 0,C 180,E1 -20072.199,E2 -20072.199} C_VEL
LIN {X 0,Y 230.939,Z 506.806,A -85,B 0,C 180,E1 -20075.238,E2 -20075.238} C_VEL
LIN {X 0,Y 233.081,Z 498.032,A -85,B 0,C 180,E1 -20077.798,E2 -20077.798} C_VEL
LIN {X 0,Y 235.594,Z 487.406,A -85,B 0,C 180,E1 -20080.311,E2 -20080.311} C_VEL
LIN {X 0,Y 238.215,Z 475.506,A -85,B 0,C 180,E1 -20082.567,E2 -20082.567} C_VEL
LIN {X 0,Y 240.471,Z 463.571,A -85,B 0,C 180,E1 -20084.384,E2 -20084.384} C_VEL
LIN {X 0,Y 242.53,Z 452.073,A -85,B 0,C 180,E1 -20085.763,E2 -20085.763} C_VEL
LIN {X 0,Y 244.368,Z 438.686,A -85,B 0,C 180,E1 -20087.037,E2 -20087.037} C_VEL
LIN {X 0,Y 245.857,Z 424.718,A -85,B 0,C 180,E1 -20088.004,E2 -20088.004} C_VEL
LIN {X 0,Y 246.85,Z 411.272,A -85,B 0,C 180,E1 -20088.632,E2 -20088.632} C_VEL
LIN {X 0,Y 250.356,Z 327.62,A -85,B 0,C 180,E1 -20090.961,E2 -20090.961} C_VEL
LIN {X 0,Y 242.807,Z 308.245,A -85,B 0,C 180,E1 -20092.656,E2 -20092.656} C_VEL
LIN {X 0,Y 238.712,Z 299.513,A -85,B 0,C 180,E1 -20093.569,E2 -20093.569} C_VEL
LIN {X 0,Y 229.624,Z 283.435,A -85,B 0,C 180,E1 -20095.623,E2 -20095.623} C_VEL
LIN {X 0,Y 228.214,Z 280.861,A -85,B 0,C 180,E1 -20095.965,E2 -20095.965} C_VEL
LIN {X 0,Y 227.94,Z 279.709,A -85,B 0,C 180,E1 -20096.064,E2 -20096.064} C_VEL
LIN {X 0,Y 227.898,Z 279.712,A -85,B 0,C 180,E1 -20100.297,E2 -20100.297} C_VEL
LIN {X 0,Y 227.879,Z 279.723,A -85,B 0,C 180,E1 -20103.719,E2 -20103.719} C_VEL
LIN {X 0,Y 227.861,Z 279.726,A -85,B 0,C 180,E1 -20108.087,E2 -20108.087} C_VEL
LIN {X 0,Y 227.916,Z 279.718,A -85,B 0,C 180,E1 -20112.717,E2 -20112.717} C_VEL
LIN {X 0,Y 227.924,Z 279.703,A -85,B 0,C 180,E1 -20117.288,E2 -20117.288} C_VEL
LIN {X 0,Y 227.862,Z 279.72,A -85,B 0,C 180,E1 -20121.916,E2 -20121.916} C_VEL
LIN {X 0,Y 227.882,Z 279.715,A -85,B 0,C 180,E1 -20126.375,E2 -20126.375} C_VEL
LIN {X 0,Y 227.911,Z 279.715,A -85,B 0,C 180,E1 -20130.44,E2 -20130.44} C_VEL
LIN {X 0,Y 227.921,Z 279.702,A -85,B 0,C 180,E1 -20134.428,E2 -20134.428} C_VEL
LIN {X 0,Y 227.955,Z 279.714,A -85,B 0,C 180,E1 -20138.289,E2 -20138.289} C_VEL
LIN {X 0,Y 228.028,Z 279.707,A -85,B 0,C 180,E1 -20142.828,E2 -20142.828} C_VEL
LIN {X 0,Y 228.065,Z 279.7,A -85,B 0,C 180,E1 -20147.545,E2 -20147.545} C_VEL
LIN {X 0,Y 228.262,Z 279.662,A -85,B 0,C 180,E1 -20151.147,E2 -20151.147} C_VEL
LIN {X 0,Y 228.319,Z 279.644,A -85,B 0,C 180,E1 -20152.93,E2 -20152.93} C_VEL
LIN {X 0,Y 228.55,Z 279.641,A -85,B 0,C 180,E1 -20158.24,E2 -20158.24} C_VEL
LIN {X 0,Y 228.55,Z 279.623,A -85,B 0,C 180,E1 -20161.764,E2 -20161.764} C_VEL
LIN {X 0,Y 228.321,Z 279.668,A -85,B 0,C 180,E1 -20167.075,E2 -20167.075} C_VEL
LIN {X 0,Y 228.137,Z 279.679,A -85,B 0,C 180,E1 -20170.715,E2 -20170.715} C_VEL
LIN {X 0,Y 228.058,Z 279.69,A -85,B 0,C 180,E1 -20174.275,E2 -20174.275} C_VEL
LIN {X 0,Y 227.964,Z 279.71,A -85,B 0,C 180,E1 -20178.389,E2 -20178.389} C_VEL
LIN {X 0,Y 227.215,Z 279.804,A -85,B 0,C 180,E1 -20179.863,E2 -20179.863} C_VEL
LIN {X 0,Y 224.293,Z 280.169,A -85,B 0,C 180,E1 -20182.267,E2 -20182.267} C_VEL
LIN {X 0,Y 221.894,Z 280.467,A -85,B 0,C 180,E1 -20184.229,E2 -20184.229} C_VEL
LIN {X 0,Y 220.928,Z 280.591,A -85,B 0,C 180,E1 -20185.753,E2 -20185.753} C_VEL
LIN {X 0,Y 220.881,Z 280.592,A -85,B 0,C 180,E1 -20186.269,E2 -20186.269} C_VEL
LIN {X 0,Y 220.84,Z 280.597,A -85,B 0,C 180,E1 -20190.77,E2 -20190.77} C_VEL
LIN {X 0,Y 220.804,Z 280.603,A -85,B 0,C 180,E1 -20194.957,E2 -20194.957} C_VEL
LIN {X 0,Y 220.809,Z 280.606,A -85,B 0,C 180,E1 -20199.539,E2 -20199.539} C_VEL
LIN {X 0,Y 220.776,Z 280.609,A -85,B 0,C 180,E1 -20204.456,E2 -20204.456} C_VEL
LIN {X 0,Y 220.796,Z 280.819,A -85,B 0,C 180,E1 -20206.432,E2 -20206.432} C_VEL
LIN {X 0,Y 222.213,Z 286.009,A -85,B 0,C 180,E1 -20208.791,E2 -20208.791} C_VEL
LIN {X 0,Y 224.358,Z 290.23,A -85,B 0,C 180,E1 -20209.346,E2 -20209.346} C_VEL
LIN {X 0,Y 231.733,Z 305.503,A -85,B 0,C 180,E1 -20211.177,E2 -20211.177} C_VEL
LIN {X 0,Y 239.498,Z 324.634,A -85,B 0,C 180,E1 -20213.055,E2 -20213.055} C_VEL
LIN {X 0,Y 241.931,Z 331.835,A -85,B 0,C 180,E1 -20213.656,E2 -20213.656} C_VEL
LIN {X 0,Y 243.673,Z 345.515,A -85,B 0,C 180,E1 -20214.366,E2 -20214.366} C_VEL
LIN {X 0,Y 240.327,Z 424.255,A -85,B 0,C 180,E1 -20216.624,E2 -20216.624} C_VEL
LIN {X 0,Y 239.237,Z 437.509,A -85,B 0,C 180,E1 -20217.268,E2 -20217.268} C_VEL
LIN {X 0,Y 237.484,Z 450.824,A -85,B 0,C 180,E1 -20218.189,E2 -20218.189} C_VEL
LIN {X 0,Y 235.262,Z 464.395,A -85,B 0,C 180,E1 -20219.48,E2 -20219.48} C_VEL
LIN {X 0,Y 232.892,Z 477.452,A -85,B 0,C 180,E1 -20221.13,E2 -20221.13} C_VEL
LIN {X 0,Y 230.886,Z 486.892,A -85,B 0,C 180,E1 -20222.588,E2 -20222.588} C_VEL
LIN {X 0,Y 228.643,Z 497.116,A -85,B 0,C 180,E1 -20224.512,E2 -20224.512} C_VEL
LIN {X 0,Y 226.25,Z 506.61,A -85,B 0,C 180,E1 -20226.669,E2 -20226.669} C_VEL
LIN {X 0,Y 223.91,Z 516.151,A -85,B 0,C 180,E1 -20229.323,E2 -20229.323} C_VEL
LIN {X 0,Y 222.064,Z 523.724,A -85,B 0,C 180,E1 -20231.904,E2 -20231.904} C_VEL
LIN {X 0,Y 220.703,Z 530.604,A -85,B 0,C 180,E1 -20234.769,E2 -20234.769} C_VEL
LIN {X 0,Y 219.461,Z 536.824,A -85,B 0,C 180,E1 -20237.986,E2 -20237.986} C_VEL
LIN {X 0,Y 218.926,Z 541.052,A -85,B 0,C 180,E1 -20240.763,E2 -20240.763} C_VEL
LIN {X 0,Y 218.569,Z 545.298,A -85,B 0,C 180,E1 -20244.464,E2 -20244.464} C_VEL
LIN {X 0,Y 218.569,Z 548.065,A -85,B 0,C 180,E1 -20248.157,E2 -20248.157} C_VEL
LIN {X 0,Y 218.65,Z 548.922,A -85,B 0,C 180,E1 -20250,E2 -20250} C_VEL
LIN {X 0,Y 218.504,Z 549.607,A -85,B 0,C 180,E1 -20253.688,E2 -20253.688} C_VEL
LIN {X 0,Y 218.687,Z 548.968,A -85,B 0,C 180,E1 -20257.385,E2 -20257.385} C_VEL
LIN {X 0,Y 219.438,Z 547.015,A -85,B 0,C 180,E1 -20261.079,E2 -20261.079} C_VEL
LIN {X 0,Y 220.888,Z 543.7,A -85,B 0,C 180,E1 -20264.746,E2 -20264.746} C_VEL
LIN {X 0,Y 223.174,Z 538.928,A -85,B 0,C 180,E1 -20268.355,E2 -20268.355} C_VEL
LIN {X 0,Y 225.337,Z 534.345,A -85,B 0,C 180,E1 -20271.018,E2 -20271.018} C_VEL
LIN {X 0,Y 228.586,Z 527.732,A -85,B 0,C 180,E1 -20274.039,E2 -20274.039} C_VEL
LIN {X 0,Y 232.464,Z 519.556,A -85,B 0,C 180,E1 -20276.967,E2 -20276.967} C_VEL
LIN {X 0,Y 236.351,Z 511.05,A -85,B 0,C 180,E1 -20279.381,E2 -20279.381} C_VEL
LIN {X 0,Y 240.601,Z 500.784,A -85,B 0,C 180,E1 -20281.72,E2 -20281.72} C_VEL
LIN {X 0,Y 244.768,Z 489.356,A -85,B 0,C 180,E1 -20283.8,E2 -20283.8} C_VEL
LIN {X 0,Y 248.578,Z 477.979,A -85,B 0,C 180,E1 -20285.421,E2 -20285.421} C_VEL
LIN {X 0,Y 252.064,Z 465.556,A -85,B 0,C 180,E1 -20286.83,E2 -20286.83} C_VEL
LIN {X 0,Y 255.363,Z 451.665,A -85,B 0,C 180,E1 -20288.008,E2 -20288.008} C_VEL
LIN {X 0,Y 257.896,Z 437.735,A -85,B 0,C 180,E1 -20288.869,E2 -20288.869} C_VEL
LIN {X 0,Y 259.624,Z 423.586,A -85,B 0,C 180,E1 -20289.471,E2 -20289.471} C_VEL
LIN {X 0,Y 263.687,Z 354.003,A -85,B 0,C 180,E1 -20291.325,E2 -20291.325} C_VEL
LIN {X 0,Y 257.643,Z 340.245,A -85,B 0,C 180,E1 -20293.342,E2 -20293.342} C_VEL
LIN {X 0,Y 250.749,Z 326.889,A -85,B 0,C 180,E1 -20295.773,E2 -20295.773} C_VEL
LIN {X 0,Y 245.075,Z 317.058,A -85,B 0,C 180,E1 -20297.941,E2 -20297.941} C_VEL
LIN {X 0,Y 238.901,Z 307.31,A -85,B 0,C 180,E1 -20300.514,E2 -20300.514} C_VEL
LIN {X 0,Y 235.083,Z 301.667,A -85,B 0,C 180,E1 -20302.26,E2 -20302.26} C_VEL
LIN {X 0,Y 230.981,Z 295.845,A -85,B 0,C 180,E1 -20304.293,E2 -20304.293} C_VEL
LIN {X 0,Y 226.275,Z 289.555,A -85,B 0,C 180,E1 -20306.868,E2 -20306.868} C_VEL
LIN {X 0,Y 222.641,Z 284.982,A -85,B 0,C 180,E1 -20309.096,E2 -20309.096} C_VEL
LIN {X 0,Y 221.93,Z 283.522,A -85,B 0,C 180,E1 -20309.686,E2 -20309.686} C_VEL
LIN {X 0,Y 220.868,Z 280.587,A -85,B 0,C 180,E1 -20312.751,E2 -20312.751} C_VEL
LIN {X 0,Y 220.877,Z 280.595,A -85,B 0,C 180,E1 -20317.551,E2 -20317.551} C_VEL
LIN {X 0,Y 220.982,Z 280.579,A -85,B 0,C 180,E1 -20322.569,E2 -20322.569} C_VEL
LIN {X 0,Y 221.009,Z 280.571,A -85,B 0,C 180,E1 -20327.136,E2 -20327.136} C_VEL
LIN {X 0,Y 221.232,Z 280.55,A -85,B 0,C 180,E1 -20330.858,E2 -20330.858} C_VEL
LIN {X 0,Y 221.284,Z 280.531,A -85,B 0,C 180,E1 -20332.699,E2 -20332.699} C_VEL
LIN {X 0,Y 221.507,Z 280.509,A -85,B 0,C 180,E1 -20338.179,E2 -20338.179} C_VEL
LIN {X 0,Y 221.507,Z 280.505,A -85,B 0,C 180,E1 -20341.816,E2 -20341.816} C_VEL
LIN {X 0,Y 221.298,Z 280.542,A -85,B 0,C 180,E1 -20347.296,E2 -20347.296} C_VEL
LIN {X 0,Y 221.105,Z 280.562,A -85,B 0,C 180,E1 -20350.992,E2 -20350.992} C_VEL
LIN {X 0,Y 221.006,Z 280.577,A -85,B 0,C 180,E1 -20356.035,E2 -20356.035} C_VEL
LIN {X 0,Y 221.788,Z 283.085,A -85,B 0,C 180,E1 -20356.703,E2 -20356.703} C_VEL
LIN {X 0,Y 223.802,Z 285.432,A -85,B 0,C 180,E1 -20358.002,E2 -20358.002} C_VEL
LIN {X 0,Y 225.616,Z 286.64,A -85,B 0,C 180,E1 -20359.03,E2 -20359.03} C_VEL
LIN {X 0,Y 227.296,Z 289.608,A -85,B 0,C 180,E1 -20360.058,E2 -20360.058} C_VEL
LIN {X 0,Y 230.061,Z 292.19,A -85,B 0,C 180,E1 -20361.502,E2 -20361.502} C_VEL
LIN {X 0,Y 232.249,Z 295.411,A -85,B 0,C 180,E1 -20362.648,E2 -20362.648} C_VEL
LIN {X 0,Y 234.256,Z 297.472,A -85,B 0,C 180,E1 -20363.596,E2 -20363.596} C_VEL
LIN {X 0,Y 237.003,Z 301.159,A -85,B 0,C 180,E1 -20364.877,E2 -20364.877} C_VEL
LIN {X 0,Y 241.599,Z 307.267,A -85,B 0,C 180,E1 -20366.856,E2 -20366.856} C_VEL
LIN {X 0,Y 247.348,Z 315.366,A -85,B 0,C 180,E1 -20369.113,E2 -20369.113} C_VEL
LIN {X 0,Y 253.998,Z 326.462,A -85,B 0,C 180,E1 -20371.539,E2 -20371.539} C_VEL
LIN {X 0,Y 260.529,Z 338.799,A -85,B 0,C 180,E1 -20373.744,E2 -20373.744} C_VEL
LIN {X 0,Y 264.1,Z 346.311,A -85,B 0,C 180,E1 -20374.896,E2 -20374.896} C_VEL
LIN {X 0,Y 260.101,Z 413.31,A -85,B 0,C 180,E1 -20376.669,E2 -20376.669} C_VEL
LIN {X 0,Y 258.456,Z 427.348,A -85,B 0,C 180,E1 -20377.288,E2 -20377.288} C_VEL
LIN {X 0,Y 255.999,Z 441.54,A -85,B 0,C 180,E1 -20378.203,E2 -20378.203} C_VEL
LIN {X 0,Y 253.416,Z 453.59,A -85,B 0,C 180,E1 -20379.269,E2 -20379.269} C_VEL
LIN {X 0,Y 250.122,Z 465.908,A -85,B 0,C 180,E1 -20380.656,E2 -20380.656} C_VEL
LIN {X 0,Y 246.291,Z 478.092,A -85,B 0,C 180,E1 -20382.41,E2 -20382.41} C_VEL
LIN {X 0,Y 242.263,Z 489.038,A -85,B 0,C 180,E1 -20384.382,E2 -20384.382} C_VEL
LIN {X 0,Y 238.149,Z 499.164,A -85,B 0,C 180,E1 -20386.677,E2 -20386.677} C_VEL
LIN {X 0,Y 234.142,Z 508.192,A -85,B 0,C 180,E1 -20389.245,E2 -20389.245} C_VEL
LIN {X 0,Y 230.585,Z 515.609,A -85,B 0,C 180,E1 -20391.889,E2 -20391.889} C_VEL
LIN {X 0,Y 227.056,Z 522.626,A -85,B 0,C 180,E1 -20395.068,E2 -20395.068} C_VEL
LIN {X 0,Y 224.532,Z 527.384,A -85,B 0,C 180,E1 -20397.853,E2 -20397.853} C_VEL
LIN {X 0,Y 222.487,Z 531.142,A -85,B 0,C 180,E1 -20400.685,E2 -20400.685} C_VEL
LIN {X 0,Y 220.903,Z 534,A -85,B 0,C 180,E1 -20403.551,E2 -20403.551} C_VEL
LIN {X 0,Y 219.432,Z 536.427,A -85,B 0,C 180,E1 -20407.398,E2 -20407.398} C_VEL
LIN {X 0,Y 218.547,Z 537.411,A -85,B 0,C 180,E1 -20411.242,E2 -20411.242} C_VEL
LIN {X 0,Y 218.281,Z 536.989,A -85,B 0,C 180,E1 -20415.074,E2 -20415.074} C_VEL
LIN {X 0,Y 218.263,Z 535.19,A -85,B 0,C 180,E1 -20418.861,E2 -20418.861} C_VEL
LIN {X 0,Y 218.754,Z 531.987,A -85,B 0,C 180,E1 -20422.617,E2 -20422.617} C_VEL
LIN {X 0,Y 219.334,Z 528.577,A -85,B 0,C 180,E1 -20425.406,E2 -20425.406} C_VEL
LIN {X 0,Y 220.412,Z 522.696,A -85,B 0,C 180,E1 -20429.087,E2 -20429.087} C_VEL
LIN {X 0,Y 221.826,Z 516.079,A -85,B 0,C 180,E1 -20432.27,E2 -20432.27} C_VEL
LIN {X 0,Y 223.859,Z 507.843,A -85,B 0,C 180,E1 -20435.404,E2 -20435.404} C_VEL
LIN {X 0,Y 226.041,Z 499.237,A -85,B 0,C 180,E1 -20438.043,E2 -20438.043} C_VEL
LIN {X 0,Y 228.611,Z 488.81,A -85,B 0,C 180,E1 -20440.629,E2 -20440.629} C_VEL
LIN {X 0,Y 231.329,Z 477.146,A -85,B 0,C 180,E1 -20442.948,E2 -20442.948} C_VEL
LIN {X 0,Y 233.676,Z 465.509,A -85,B 0,C 180,E1 -20444.812,E2 -20444.812} C_VEL
LIN {X 0,Y 235.654,Z 454.469,A -85,B 0,C 180,E1 -20446.236,E2 -20446.236} C_VEL
LIN {X 0,Y 237.627,Z 441.657,A -85,B 0,C 180,E1 -20447.536,E2 -20447.536} C_VEL
LIN {X 0,Y 239.3,Z 427.249,A -85,B 0,C 180,E1 -20448.626,E2 -20448.626} C_VEL
LIN {X 0,Y 240.489,Z 412.822,A -85,B 0,C 180,E1 -20449.36,E2 -20449.36} C_VEL
LIN {X 0,Y 244.24,Z 329.895,A -85,B 0,C 180,E1 -20451.714,E2 -20451.714} C_VEL
LIN {X 0,Y 239.553,Z 317.234,A -85,B 0,C 180,E1 -20452.82,E2 -20452.82} C_VEL
LIN {X 0,Y 234.158,Z 304.716,A -85,B 0,C 180,E1 -20454.09,E2 -20454.09} C_VEL
LIN {X 0,Y 226.17,Z 290.443,A -85,B 0,C 180,E1 -20455.956,E2 -20455.956} C_VEL
LIN {X 0,Y 222.833,Z 284.672,A -85,B 0,C 180,E1 -20456.776,E2 -20456.776} C_VEL
LIN {X 0,Y 221.199,Z 282.053,A -85,B 0,C 180,E1 -20457.181,E2 -20457.181} C_VEL
LIN {X 0,Y 220.841,Z 280.601,A -85,B 0,C 180,E1 -20457.324,E2 -20457.324} C_VEL
LIN {X 0,Y 220.853,Z 280.593,A -85,B 0,C 180,E1 -20460.78,E2 -20460.78} C_VEL
LIN {X 0,Y 220.805,Z 280.606,A -85,B 0,C 180,E1 -20464.954,E2 -20464.954} C_VEL
LIN {X 0,Y 220.848,Z 280.59,A -85,B 0,C 180,E1 -20469.527,E2 -20469.527} C_VEL
LIN {X 0,Y 220.875,Z 280.596,A -85,B 0,C 180,E1 -20472.964,E2 -20472.964} C_VEL
LIN {X 0,Y 220.881,Z 280.579,A -85,B 0,C 180,E1 -20477.038,E2 -20477.038} C_VEL
LIN {X 0,Y 220.851,Z 280.598,A -85,B 0,C 180,E1 -20480.476,E2 -20480.476} C_VEL
LIN {X 0,Y 220.807,Z 280.584,A -85,B 0,C 180,E1 -20485.05,E2 -20485.05} C_VEL
LIN {X 0,Y 220.86,Z 280.595,A -85,B 0,C 180,E1 -20489.397,E2 -20489.397} C_VEL
LIN {X 0,Y 220.888,Z 280.571,A -85,B 0,C 180,E1 -20493.552,E2 -20493.552} C_VEL
LIN {X 0,Y 220.871,Z 280.597,A -85,B 0,C 180,E1 -20497.556,E2 -20497.556} C_VEL
LIN {X 0,Y 220.978,Z 280.584,A -85,B 0,C 180,E1 -20502.574,E2 -20502.574} C_VEL
LIN {X 0,Y 221.005,Z 280.58,A -85,B 0,C 180,E1 -20507.141,E2 -20507.141} C_VEL
LIN {X 0,Y 221.199,Z 280.543,A -85,B 0,C 180,E1 -20510.862,E2 -20510.862} C_VEL
LIN {X 0,Y 221.254,Z 280.523,A -85,B 0,C 180,E1 -20512.703,E2 -20512.703} C_VEL
LIN {X 0,Y 221.508,Z 280.518,A -85,B 0,C 180,E1 -20518.184,E2 -20518.184} C_VEL
LIN {X 0,Y 221.508,Z 280.498,A -85,B 0,C 180,E1 -20521.821,E2 -20521.821} C_VEL
LIN {X 0,Y 221.256,Z 280.548,A -85,B 0,C 180,E1 -20527.302,E2 -20527.302} C_VEL
LIN {X 0,Y 221.065,Z 280.559,A -85,B 0,C 180,E1 -20530.999,E2 -20530.999} C_VEL
LIN {X 0,Y 221.013,Z 280.58,A -85,B 0,C 180,E1 -20536.632,E2 -20536.632} C_VEL
LIN {X 0,Y 220.883,Z 280.596,A -85,B 0,C 180,E1 -20540.489,E2 -20540.489} C_VEL
LIN {X 0,Y 220.862,Z 280.597,A -85,B 0,C 180,E1 -20544.438,E2 -20544.438} C_VEL
LIN {X 0,Y 220.881,Z 280.592,A -85,B 0,C 180,E1 -20546.269,E2 -20546.269} C_VEL
LIN {X 0,Y 220.277,Z 280.675,A -85,B 0,C 180,E1 -20547.791,E2 -20547.791} C_VEL
LIN {X 0,Y 218.691,Z 280.875,A -85,B 0,C 180,E1 -20549.286,E2 -20549.286} C_VEL
LIN {X 0,Y 214.89,Z 281.344,A -85,B 0,C 180,E1 -20552.301,E2 -20552.301} C_VEL
LIN {X 0,Y 213.837,Z 281.473,A -85,B 0,C 180,E1 -20553.879,E2 -20553.879} C_VEL
LIN {X 0,Y 213.764,Z 281.48,A -85,B 0,C 180,E1 -20554.415,E2 -20554.415} C_VEL
LIN {X 0,Y 213.726,Z 281.488,A -85,B 0,C 180,E1 -20558.669,E2 -20558.669} C_VEL
LIN {X 0,Y 213.715,Z 281.488,A -85,B 0,C 180,E1 -20561.127,E2 -20561.127} C_VEL
LIN {X 0,Y 213.752,Z 281.646,A -85,B 0,C 180,E1 -20565.404,E2 -20565.404} C_VEL
LIN {X 0,Y 214.895,Z 285.918,A -85,B 0,C 180,E1 -20567.38,E2 -20567.38} C_VEL
LIN {X 0,Y 223.745,Z 303.279,A -85,B 0,C 180,E1 -20569.742,E2 -20569.742} C_VEL
LIN {X 0,Y 230.496,Z 318.978,A -85,B 0,C 180,E1 -20571.473,E2 -20571.473} C_VEL
LIN {X 0,Y 235.837,Z 333.137,A -85,B 0,C 180,E1 -20572.813,E2 -20572.813} C_VEL
LIN {X 0,Y 237.527,Z 346.871,A -85,B 0,C 180,E1 -20573.544,E2 -20573.544} C_VEL
LIN {X 0,Y 234.096,Z 424.164,A -85,B 0,C 180,E1 -20575.808,E2 -20575.808} C_VEL
LIN {X 0,Y 232.886,Z 438.163,A -85,B 0,C 180,E1 -20576.518,E2 -20576.518} C_VEL
LIN {X 0,Y 230.864,Z 452.378,A -85,B 0,C 180,E1 -20577.552,E2 -20577.552} C_VEL
LIN {X 0,Y 228.775,Z 464.681,A -85,B 0,C 180,E1 -20578.775,E2 -20578.775} C_VEL
LIN {X 0,Y 226.35,Z 477.483,A -85,B 0,C 180,E1 -20580.44,E2 -20580.44} C_VEL
LIN {X 0,Y 224.258,Z 487.018,A -85,B 0,C 180,E1 -20581.961,E2 -20581.961} C_VEL
LIN {X 0,Y 221.651,Z 498.186,A -85,B 0,C 180,E1 -20584.153,E2 -20584.153} C_VEL
LIN {X 0,Y 219.227,Z 507.506,A -85,B 0,C 180,E1 -20586.377,E2 -20586.377} C_VEL
LIN {X 0,Y 216.845,Z 516.837,A -85,B 0,C 180,E1 -20589.114,E2 -20589.114} C_VEL
LIN {X 0,Y 214.808,Z 525.334,A -85,B 0,C 180,E1 -20592.211,E2 -20592.211} C_VEL
LIN {X 0,Y 213.166,Z 532.903,A -85,B 0,C 180,E1 -20595.684,E2 -20595.684} C_VEL
LIN {X 0,Y 211.999,Z 539.312,A -85,B 0,C 180,E1 -20599.494,E2 -20599.494} C_VEL
LIN {X 0,Y 211.623,Z 542.972,A -85,B 0,C 180,E1 -20602.366,E2 -20602.366} C_VEL
LIN {X 0,Y 211.423,Z 546.527,A -85,B 0,C 180,E1 -20606.188,E2 -20606.188} C_VEL
LIN {X 0,Y 211.566,Z 548.65,A -85,B 0,C 180,E1 -20610,E2 -20610} C_VEL
LIN {X 0,Y 211.403,Z 549.391,A -85,B 0,C 180,E1 -20613.812,E2 -20613.812} C_VEL
LIN {X 0,Y 211.627,Z 548.811,A -85,B 0,C 180,E1 -20617.633,E2 -20617.633} C_VEL
LIN {X 0,Y 212.425,Z 546.922,A -85,B 0,C 180,E1 -20621.449,E2 -20621.449} C_VEL
LIN {X 0,Y 214.012,Z 543.685,A -85,B 0,C 180,E1 -20625.231,E2 -20625.231} C_VEL
LIN {X 0,Y 216.414,Z 538.991,A -85,B 0,C 180,E1 -20628.95,E2 -20628.95} C_VEL
LIN {X 0,Y 218.707,Z 534.447,A -85,B 0,C 180,E1 -20631.687,E2 -20631.687} C_VEL
LIN {X 0,Y 222.117,Z 527.911,A -85,B 0,C 180,E1 -20634.786,E2 -20634.786} C_VEL
LIN {X 0,Y 226.151,Z 519.846,A -85,B 0,C 180,E1 -20637.784,E2 -20637.784} C_VEL
LIN {X 0,Y 230.191,Z 511.428,A -85,B 0,C 180,E1 -20640.248,E2 -20640.248} C_VEL
LIN {X 0,Y 234.625,Z 501.312,A -85,B 0,C 180,E1 -20642.626,E2 -20642.626} C_VEL
LIN {X 0,Y 238.932,Z 490.035,A -85,B 0,C 180,E1 -20644.742,E2 -20644.742} C_VEL
LIN {X 0,Y 242.88,Z 478.843,A -85,B 0,C 180,E1 -20646.383,E2 -20646.383} C_VEL
LIN {X 0,Y 246.473,Z 466.674,A -85,B 0,C 180,E1 -20647.81,E2 -20647.81} C_VEL
LIN {X 0,Y 249.886,Z 453.146,A -85,B 0,C 180,E1 -20648.997,E2 -20648.997} C_VEL
LIN {X 0,Y 252.559,Z 439.077,A -85,B 0,C 180,E1 -20649.916,E2 -20649.916} C_VEL
LIN {X 0,Y 254.468,Z 424.87,A -85,B 0,C 180,E1 -20650.546,E2 -20650.546} C_VEL
LIN {X 0,Y 256.336,Z 397.288,A -85,B 0,C 180,E1 -20651.31,E2 -20651.31} C_VEL
LIN {X 0,Y 258.71,Z 356.383,A -85,B 0,C 180,E1 -20652.407,E2 -20652.407} C_VEL
LIN {X 0,Y 252.617,Z 342.65,A -85,B 0,C 180,E1 -20654.552,E2 -20654.552} C_VEL
LIN {X 0,Y 246.999,Z 331.639,A -85,B 0,C 180,E1 -20656.649,E2 -20656.649} C_VEL
LIN {X 0,Y 241.844,Z 322.462,A -85,B 0,C 180,E1 -20658.715,E2 -20658.715} C_VEL
LIN {X 0,Y 235.857,Z 312.795,A -85,B 0,C 180,E1 -20661.335,E2 -20661.335} C_VEL
LIN {X 0,Y 232.047,Z 307.025,A -85,B 0,C 180,E1 -20663.166,E2 -20663.166} C_VEL
LIN {X 0,Y 228.368,Z 301.754,A -85,B 0,C 180,E1 -20665.076,E2 -20665.076} C_VEL
LIN {X 0,Y 224.005,Z 295.723,A -85,B 0,C 180,E1 -20667.576,E2 -20667.576} C_VEL
LIN {X 0,Y 220.542,Z 291.194,A -85,B 0,C 180,E1 -20669.806,E2 -20669.806} C_VEL
LIN {X 0,Y 219.708,Z 289.851,A -85,B 0,C 180,E1 -20670.406,E2 -20670.406} C_VEL
LIN {X 0,Y 216.595,Z 286.409,A -85,B 0,C 180,E1 -20672.691,E2 -20672.691} C_VEL
LIN {X 0,Y 214.434,Z 283.575,A -85,B 0,C 180,E1 -20674.519,E2 -20674.519} C_VEL
LIN {X 0,Y 214.117,Z 282.838,A -85,B 0,C 180,E1 -20674.999,E2 -20674.999} C_VEL
LIN {X 0,Y 213.846,Z 281.463,A -85,B 0,C 180,E1 -20676.77,E2 -20676.77} C_VEL
LIN {X 0,Y 213.941,Z 281.453,A -85,B 0,C 180,E1 -20682.801,E2 -20682.801} C_VEL
LIN {X 0,Y 213.95,Z 281.455,A -85,B 0,C 180,E1 -20686.704,E2 -20686.704} C_VEL
LIN {X 0,Y 214.164,Z 281.434,A -85,B 0,C 180,E1 -20690.554,E2 -20690.554} C_VEL
LIN {X 0,Y 214.222,Z 281.411,A -85,B 0,C 180,E1 -20692.457,E2 -20692.457} C_VEL
LIN {X 0,Y 214.44,Z 281.389,A -85,B 0,C 180,E1 -20698.119,E2 -20698.119} C_VEL
LIN {X 0,Y 214.549,Z 281.378,A -85,B 0,C 180,E1 -20699.997,E2 -20699.997} C_VEL
LIN {X 0,Y 214.44,Z 281.385,A -85,B 0,C 180,E1 -20701.876,E2 -20701.876} C_VEL
LIN {X 0,Y 214.233,Z 281.425,A -85,B 0,C 180,E1 -20707.538,E2 -20707.538} C_VEL
LIN {X 0,Y 214.065,Z 281.596,A -85,B 0,C 180,E1 -20711.418,E2 -20711.418} C_VEL
LIN {X 0,Y 214.621,Z 283.565,A -85,B 0,C 180,E1 -20712.047,E2 -20712.047} C_VEL
LIN {X 0,Y 216.315,Z 285.923,A -85,B 0,C 180,E1 -20713.502,E2 -20713.502} C_VEL
LIN {X 0,Y 218.934,Z 287.489,A -85,B 0,C 180,E1 -20715.354,E2 -20715.354} C_VEL
LIN {X 0,Y 220.429,Z 290.396,A -85,B 0,C 180,E1 -20716.494,E2 -20716.494} C_VEL
LIN {X 0,Y 223.007,Z 292.72,A -85,B 0,C 180,E1 -20718.115,E2 -20718.115} C_VEL
LIN {X 0,Y 223.828,Z 293.902,A -85,B 0,C 180,E1 -20718.63,E2 -20718.63} C_VEL
LIN {X 0,Y 226.124,Z 296.962,A -85,B 0,C 180,E1 -20719.989,E2 -20719.989} C_VEL
LIN {X 0,Y 227.9,Z 298.778,A -85,B 0,C 180,E1 -20720.946,E2 -20720.946} C_VEL
LIN {X 0,Y 230.485,Z 302.244,A -85,B 0,C 180,E1 -20722.314,E2 -20722.314} C_VEL
LIN {X 0,Y 231.894,Z 303.837,A -85,B 0,C 180,E1 -20723.007,E2 -20723.007} C_VEL
LIN {X 0,Y 235.956,Z 309.337,A -85,B 0,C 180,E1 -20724.936,E2 -20724.936} C_VEL
LIN {X 0,Y 241.42,Z 316.842,A -85,B 0,C 180,E1 -20727.287,E2 -20727.287} C_VEL
LIN {X 0,Y 246.123,Z 324.08,A -85,B 0,C 180,E1 -20729.155,E2 -20729.155} C_VEL
LIN {X 0,Y 252.581,Z 335.702,A -85,B 0,C 180,E1 -20731.561,E2 -20731.561} C_VEL
LIN {X 0,Y 257.963,Z 346.354,A -85,B 0,C 180,E1 -20733.422,E2 -20733.422} C_VEL
LIN {X 0,Y 259.163,Z 349.017,A -85,B 0,C 180,E1 -20733.829,E2 -20733.829} C_VEL
LIN {X 0,Y 255.135,Z 413.327,A -85,B 0,C 180,E1 -20735.539,E2 -20735.539} C_VEL
LIN {X 0,Y 253.413,Z 427.615,A -85,B 0,C 180,E1 -20736.175,E2 -20736.175} C_VEL
LIN {X 0,Y 250.963,Z 441.258,A -85,B 0,C 180,E1 -20737.051,E2 -20737.051} C_VEL
LIN {X 0,Y 248.265,Z 453.346,A -85,B 0,C 180,E1 -20738.113,E2 -20738.113} C_VEL
LIN {X 0,Y 244.871,Z 465.792,A -85,B 0,C 180,E1 -20739.528,E2 -20739.528} C_VEL
LIN {X 0,Y 240.898,Z 478.034,A -85,B 0,C 180,E1 -20741.304,E2 -20741.304} C_VEL
LIN {X 0,Y 237.097,Z 488.023,A -85,B 0,C 180,E1 -20743.097,E2 -20743.097} C_VEL
LIN {X 0,Y 232.71,Z 498.326,A -85,B 0,C 180,E1 -20745.401,E2 -20745.401} C_VEL
LIN {X 0,Y 228.499,Z 507.533,A -85,B 0,C 180,E1 -20748.014,E2 -20748.014} C_VEL
LIN {X 0,Y 224.675,Z 515.1,A -85,B 0,C 180,E1 -20750.697,E2 -20750.697} C_VEL
LIN {X 0,Y 220.902,Z 522.263,A -85,B 0,C 180,E1 -20753.945,E2 -20753.945} C_VEL
LIN {X 0,Y 218.137,Z 527.267,A -85,B 0,C 180,E1 -20756.89,E2 -20756.89} C_VEL
LIN {X 0,Y 215.331,Z 532.103,A -85,B 0,C 180,E1 -20760.689,E2 -20760.689} C_VEL
LIN {X 0,Y 214.244,Z 533.966,A -85,B 0,C 180,E1 -20762.662,E2 -20762.662} C_VEL
LIN {X 0,Y 212.556,Z 536.505,A -85,B 0,C 180,E1 -20766.624,E2 -20766.624} C_VEL
LIN {X 0,Y 211.558,Z 537.591,A -85,B 0,C 180,E1 -20770.598,E2 -20770.598} C_VEL
LIN {X 0,Y 211.185,Z 537.271,A -85,B 0,C 180,E1 -20774.561,E2 -20774.561} C_VEL
LIN {X 0,Y 211.143,Z 535.571,A -85,B 0,C 180,E1 -20778.48,E2 -20778.48} C_VEL
LIN {X 0,Y 211.6,Z 532.469,A -85,B 0,C 180,E1 -20782.366,E2 -20782.366} C_VEL
LIN {X 0,Y 212.201,Z 529.164,A -85,B 0,C 180,E1 -20785.251,E2 -20785.251} C_VEL
LIN {X 0,Y 213.271,Z 523.396,A -85,B 0,C 180,E1 -20789.056,E2 -20789.056} C_VEL
LIN {X 0,Y 214.697,Z 516.904,A -85,B 0,C 180,E1 -20792.345,E2 -20792.345} C_VEL
LIN {X 0,Y 216.777,Z 508.839,A -85,B 0,C 180,E1 -20795.582,E2 -20795.582} C_VEL
LIN {X 0,Y 219.023,Z 500.391,A -85,B 0,C 180,E1 -20798.302,E2 -20798.302} C_VEL
LIN {X 0,Y 221.646,Z 490.209,A -85,B 0,C 180,E1 -20800.967,E2 -20800.967} C_VEL
LIN {X 0,Y 224.455,Z 478.785,A -85,B 0,C 180,E1 -20803.351,E2 -20803.351} C_VEL
LIN {X 0,Y 226.894,Z 467.448,A -85,B 0,C 180,E1 -20805.265,E2 -20805.265} C_VEL
LIN {X 0,Y 228.822,Z 456.854,A -85,B 0,C 180,E1 -20806.735,E2 -20806.735} C_VEL
LIN {X 0,Y 230.941,Z 444.603,A -85,B 0,C 180,E1 -20808.061,E2 -20808.061} C_VEL
LIN {X 0,Y 232.709,Z 430.406,A -85,B 0,C 180,E1 -20809.231,E2 -20809.231} C_VEL
LIN {X 0,Y 234.022,Z 416.294,A -85,B 0,C 180,E1 -20810.032,E2 -20810.032} C_VEL
LIN {X 0,Y 235.029,Z 396.961,A -85,B 0,C 180,E1 -20810.684,E2 -20810.684} C_VEL
LIN {X 0,Y 238.105,Z 331.509,A -85,B 0,C 180,E1 -20812.533,E2 -20812.533} C_VEL
LIN {X 0,Y 231.791,Z 314.928,A -85,B 0,C 180,E1 -20814.095,E2 -20814.095} C_VEL
LIN {X 0,Y 228.062,Z 306.95,A -85,B 0,C 180,E1 -20815.003,E2 -20815.003} C_VEL
LIN {X 0,Y 219.556,Z 291.821,A -85,B 0,C 180,E1 -20817.099,E2 -20817.099} C_VEL
LIN {X 0,Y 215.627,Z 285.436,A -85,B 0,C 180,E1 -20818.115,E2 -20818.115} C_VEL
LIN {X 0,Y 214.078,Z 282.799,A -85,B 0,C 180,E1 -20818.535,E2 -20818.535} C_VEL
LIN {X 0,Y 213.798,Z 281.469,A -85,B 0,C 180,E1 -20818.702,E2 -20818.702} C_VEL
LIN {X 0,Y 213.769,Z 281.482,A -85,B 0,C 180,E1 -20821.737,E2 -20821.737} C_VEL
LIN {X 0,Y 213.745,Z 281.481,A -85,B 0,C 180,E1 -20826.287,E2 -20826.287} C_VEL
LIN {X 0,Y 213.789,Z 281.467,A -85,B 0,C 180,E1 -20831.106,E2 -20831.106} C_VEL
LIN {X 0,Y 213.827,Z 281.474,A -85,B 0,C 180,E1 -20833.694,E2 -20833.694} C_VEL
LIN {X 0,Y 213.831,Z 281.457,A -85,B 0,C 180,E1 -20836.358,E2 -20836.358} C_VEL
LIN {X 0,Y 213.815,Z 281.471,A -85,B 0,C 180,E1 -20839.112,E2 -20839.112} C_VEL
LIN {X 0,Y 213.746,Z 281.461,A -85,B 0,C 180,E1 -20843.716,E2 -20843.716} C_VEL
LIN {X 0,Y 213.788,Z 281.479,A -85,B 0,C 180,E1 -20848.727,E2 -20848.727} C_VEL
LIN {X 0,Y 213.819,Z 281.45,A -85,B 0,C 180,E1 -20852.605,E2 -20852.605} C_VEL
LIN {X 0,Y 213.845,Z 281.471,A -85,B 0,C 180,E1 -20856.955,E2 -20856.955} C_VEL
LIN {X 0,Y 213.956,Z 281.46,A -85,B 0,C 180,E1 -20862.808,E2 -20862.808} C_VEL
LIN {X 0,Y 213.946,Z 281.457,A -85,B 0,C 180,E1 -20866.709,E2 -20866.709} C_VEL
LIN {X 0,Y 214.136,Z 281.424,A -85,B 0,C 180,E1 -20870.558,E2 -20870.558} C_VEL
LIN {X 0,Y 214.096,Z 281.419,A -85,B 0,C 180,E1 -20874.351,E2 -20874.351} C_VEL
LIN {X 0,Y 214.441,Z 281.398,A -85,B 0,C 180,E1 -20878.124,E2 -20878.124} C_VEL
LIN {X 0,Y 214.546,Z 281.379,A -85,B 0,C 180,E1 -20880.003,E2 -20880.003} C_VEL
LIN {X 0,Y 214.441,Z 281.376,A -85,B 0,C 180,E1 -20881.881,E2 -20881.881} C_VEL
LIN {X 0,Y 214.196,Z 281.428,A -85,B 0,C 180,E1 -20887.544,E2 -20887.544} C_VEL
LIN {X 0,Y 213.997,Z 281.435,A -85,B 0,C 180,E1 -20891.367,E2 -20891.367} C_VEL
LIN {X 0,Y 213.928,Z 281.457,A -85,B 0,C 180,E1 -20895.24,E2 -20895.24} C_VEL
LIN {X 0,Y 213.834,Z 281.467,A -85,B 0,C 180,E1 -20899.19,E2 -20899.19} C_VEL
LIN {X 0,Y 213.811,Z 281.472,A -85,B 0,C 180,E1 -20903.234,E2 -20903.234} C_VEL
LIN {X 0,Y 213.831,Z 281.47,A -85,B 0,C 180,E1 -20907.452,E2 -20907.452} C_VEL
LIN {X 0,Y 213.77,Z 281.479,A -85,B 0,C 180,E1 -20911.74,E2 -20911.74} C_VEL
LIN {X 0,Y 213.764,Z 281.48,A -85,B 0,C 180,E1 -20914.415,E2 -20914.415} C_VEL
LIN {X 0,Y 213.464,Z 281.519,A -85,B 0,C 180,E1 -20915.466,E2 -20915.466} C_VEL
LIN {X 0,Y 212.112,Z 281.69,A -85,B 0,C 180,E1 -20917.019,E2 -20917.019} C_VEL
LIN {X 0,Y 207.735,Z 282.232,A -85,B 0,C 180,E1 -20920.648,E2 -20920.648} C_VEL
LIN {X 0,Y 206.697,Z 282.362,A -85,B 0,C 180,E1 -20922.28,E2 -20922.28} C_VEL
LIN {X 0,Y 206.626,Z 282.369,A -85,B 0,C 180,E1 -20922.833,E2 -20922.833} C_VEL
LIN {X 0,Y 206.681,Z 282.423,A -85,B 0,C 180,E1 -20924.27,E2 -20924.27} C_VEL
LIN {X 0,Y 207.608,Z 285.712,A -85,B 0,C 180,E1 -20925.857,E2 -20925.857} C_VEL
LIN {X 0,Y 209.921,Z 290.004,A -85,B 0,C 180,E1 -20926.536,E2 -20926.536} C_VEL
LIN {X 0,Y 218.484,Z 306.886,A -85,B 0,C 180,E1 -20928.929,E2 -20928.929} C_VEL
LIN {X 0,Y 224.961,Z 322.063,A -85,B 0,C 180,E1 -20930.674,E2 -20930.674} C_VEL
LIN {X 0,Y 230.101,Z 336.098,A -85,B 0,C 180,E1 -20932.038,E2 -20932.038} C_VEL
LIN {X 0,Y 231.44,Z 347.742,A -85,B 0,C 180,E1 -20932.671,E2 -20932.671} C_VEL
LIN {X 0,Y 227.925,Z 423.945,A -85,B 0,C 180,E1 -20934.95,E2 -20934.95} C_VEL
LIN {X 0,Y 226.657,Z 437.952,A -85,B 0,C 180,E1 -20935.672,E2 -20935.672} C_VEL
LIN {X 0,Y 224.692,Z 451.611,A -85,B 0,C 180,E1 -20936.68,E2 -20936.68} C_VEL
LIN {X 0,Y 222.326,Z 464.926,A -85,B 0,C 180,E1 -20938.03,E2 -20938.03} C_VEL
LIN {X 0,Y 219.85,Z 477.489,A -85,B 0,C 180,E1 -20939.711,E2 -20939.711} C_VEL
LIN {X 0,Y 217.657,Z 487.124,A -85,B 0,C 180,E1 -20941.295,E2 -20941.295} C_VEL
LIN {X 0,Y 215.262,Z 497.26,A -85,B 0,C 180,E1 -20943.326,E2 -20943.326} C_VEL
LIN {X 0,Y 212.659,Z 506.685,A -85,B 0,C 180,E1 -20945.6,E2 -20945.6} C_VEL
LIN {X 0,Y 210.15,Z 516.132,A -85,B 0,C 180,E1 -20948.416,E2 -20948.416} C_VEL
LIN {X 0,Y 208.102,Z 523.809,A -85,B 0,C 180,E1 -20951.217,E2 -20951.217} C_VEL
LIN {X 0,Y 206.675,Z 530.485,A -85,B 0,C 180,E1 -20954.214,E2 -20954.214} C_VEL
LIN {X 0,Y 205.471,Z 535.828,A -85,B 0,C 180,E1 -20957.154,E2 -20957.154} C_VEL
LIN {X 0,Y 204.67,Z 541.453,A -85,B 0,C 180,E1 -20961.111,E2 -20961.111} C_VEL
LIN {X 0,Y 204.396,Z 544.571,A -85,B 0,C 180,E1 -20964.079,E2 -20964.079} C_VEL
LIN {X 0,Y 204.37,Z 547.46,A -85,B 0,C 180,E1 -20968.029,E2 -20968.029} C_VEL
LIN {X 0,Y 204.483,Z 548.378,A -85,B 0,C 180,E1 -20970,E2 -20970} C_VEL
LIN {X 0,Y 204.303,Z 549.176,A -85,B 0,C 180,E1 -20973.945,E2 -20973.945} C_VEL
LIN {X 0,Y 204.564,Z 548.655,A -85,B 0,C 180,E1 -20977.898,E2 -20977.898} C_VEL
LIN {X 0,Y 205.431,Z 546.826,A -85,B 0,C 180,E1 -20981.845,E2 -20981.845} C_VEL
LIN {X 0,Y 207.124,Z 543.659,A -85,B 0,C 180,E1 -20985.75,E2 -20985.75} C_VEL
LIN {X 0,Y 209.676,Z 539.057,A -85,B 0,C 180,E1 -20989.583,E2 -20989.583} C_VEL
LIN {X 0,Y 213.028,Z 532.851,A -85,B 0,C 180,E1 -20993.321,E2 -20993.321} C_VEL
LIN {X 0,Y 216.816,Z 525.975,A -85,B 0,C 180,E1 -20996.467,E2 -20996.467} C_VEL
LIN {X 0,Y 221.239,Z 517.481,A -85,B 0,C 180,E1 -20999.496,E2 -20999.496} C_VEL
LIN {X 0,Y 225.595,Z 508.642,A -85,B 0,C 180,E1 -21001.978,E2 -21001.978} C_VEL
LIN {X 0,Y 230.156,Z 498.321,A -85,B 0,C 180,E1 -21004.303,E2 -21004.303} C_VEL
LIN {X 0,Y 234.048,Z 488.404,A -85,B 0,C 180,E1 -21006.106,E2 -21006.106} C_VEL
LIN {X 0,Y 238.179,Z 476.914,A -85,B 0,C 180,E1 -21007.753,E2 -21007.753} C_VEL
LIN {X 0,Y 241.953,Z 464.338,A -85,B 0,C 180,E1 -21009.18,E2 -21009.18} C_VEL
LIN {X 0,Y 245.227,Z 451.346,A -85,B 0,C 180,E1 -21010.286,E2 -21010.286} C_VEL
LIN {X 0,Y 247.916,Z 437.394,A -85,B 0,C 180,E1 -21011.162,E2 -21011.162} C_VEL
LIN {X 0,Y 249.812,Z 422.758,A -85,B 0,C 180,E1 -21011.789,E2 -21011.789} C_VEL
LIN {X 0,Y 253.874,Z 359.058,A -85,B 0,C 180,E1 -21013.51,E2 -21013.51} C_VEL
LIN {X 0,Y 248.578,Z 346.896,A -85,B 0,C 180,E1 -21015.479,E2 -21015.479} C_VEL
LIN {X 0,Y 242.972,Z 335.752,A -85,B 0,C 180,E1 -21017.689,E2 -21017.689} C_VEL
LIN {X 0,Y 238.488,Z 327.586,A -85,B 0,C 180,E1 -21019.583,E2 -21019.583} C_VEL
LIN {X 0,Y 233.02,Z 318.476,A -85,B 0,C 180,E1 -21022.106,E2 -21022.106} C_VEL
LIN {X 0,Y 229.416,Z 312.95,A -85,B 0,C 180,E1 -21023.913,E2 -21023.913} C_VEL
LIN {X 0,Y 225.87,Z 307.654,A -85,B 0,C 180,E1 -21025.844,E2 -21025.844} C_VEL
LIN {X 0,Y 222,Z 302.152,A -85,B 0,C 180,E1 -21028.158,E2 -21028.158} C_VEL
LIN {X 0,Y 218.403,Z 297.235,A -85,B 0,C 180,E1 -21030.588,E2 -21030.588} C_VEL
LIN {X 0,Y 217.205,Z 295.773,A -85,B 0,C 180,E1 -21031.458,E2 -21031.458} C_VEL
LIN {X 0,Y 212.652,Z 289.889,A -85,B 0,C 180,E1 -21035.271,E2 -21035.271} C_VEL
LIN {X 0,Y 211.019,Z 287.965,A -85,B 0,C 180,E1 -21036.868,E2 -21036.868} C_VEL
LIN {X 0,Y 208.267,Z 285.923,A -85,B 0,C 180,E1 -21039.89,E2 -21039.89} C_VEL
LIN {X 0,Y 207.093,Z 283.525,A -85,B 0,C 180,E1 -21041.684,E2 -21041.684} C_VEL
LIN {X 0,Y 206.88,Z 282.339,A -85,B 0,C 180,E1 -21042.195,E2 -21042.195} C_VEL
LIN {X 0,Y 206.892,Z 282.34,A -85,B 0,C 180,E1 -21046.242,E2 -21046.242} C_VEL
LIN {X 0,Y 207.102,Z 282.312,A -85,B 0,C 180,E1 -21050.229,E2 -21050.229} C_VEL
LIN {X 0,Y 207.163,Z 282.29,A -85,B 0,C 180,E1 -21052.198,E2 -21052.198} C_VEL
LIN {X 0,Y 207.377,Z 282.267,A -85,B 0,C 180,E1 -21058.055,E2 -21058.055} C_VEL
LIN {X 0,Y 207.514,Z 282.254,A -85,B 0,C 180,E1 -21059.997,E2 -21059.997} C_VEL
LIN {X 0,Y 207.377,Z 282.265,A -85,B 0,C 180,E1 -21061.939,E2 -21061.939} C_VEL
LIN {X 0,Y 207.09,Z 282.431,A -85,B 0,C 180,E1 -21064.559,E2 -21064.559} C_VEL
LIN {X 0,Y 207.574,Z 284.174,A -85,B 0,C 180,E1 -21065.462,E2 -21065.462} C_VEL
LIN {X 0,Y 209.184,Z 286.424,A -85,B 0,C 180,E1 -21067.599,E2 -21067.599} C_VEL
LIN {X 0,Y 212.075,Z 288.239,A -85,B 0,C 180,E1 -21070.503,E2 -21070.503} C_VEL
LIN {X 0,Y 212.522,Z 289.059,A -85,B 0,C 180,E1 -21070.961,E2 -21070.961} C_VEL
LIN {X 0,Y 213.927,Z 291.685,A -85,B 0,C 180,E1 -21072.327,E2 -21072.327} C_VEL
LIN {X 0,Y 216.481,Z 293.831,A -85,B 0,C 180,E1 -21074.329,E2 -21074.329} C_VEL
LIN {X 0,Y 217.157,Z 294.416,A -85,B 0,C 180,E1 -21074.823,E2 -21074.823} C_VEL
LIN {X 0,Y 219.214,Z 297.678,A -85,B 0,C 180,E1 -21076.364,E2 -21076.364} C_VEL
LIN {X 0,Y 221.478,Z 299.771,A -85,B 0,C 180,E1 -21077.814,E2 -21077.814} C_VEL
LIN {X 0,Y 223.873,Z 303.215,A -85,B 0,C 180,E1 -21079.31,E2 -21079.31} C_VEL
LIN {X 0,Y 225.596,Z 304.995,A -85,B 0,C 180,E1 -21080.275,E2 -21080.275} C_VEL
LIN {X 0,Y 228.524,Z 308.831,A -85,B 0,C 180,E1 -21081.869,E2 -21081.869} C_VEL
LIN {X 0,Y 233.373,Z 315.38,A -85,B 0,C 180,E1 -21084.281,E2 -21084.281} C_VEL
LIN {X 0,Y 238.918,Z 323.265,A -85,B 0,C 180,E1 -21086.768,E2 -21086.768} C_VEL
LIN {X 0,Y 243.097,Z 329.902,A -85,B 0,C 180,E1 -21088.492,E2 -21088.492} C_VEL
LIN {X 0,Y 249.182,Z 341.149,A -85,B 0,C 180,E1 -21090.859,E2 -21090.859} C_VEL
LIN {X 0,Y 254.201,Z 351.5,A -85,B 0,C 180,E1 -21092.68,E2 -21092.68} C_VEL
LIN {X 0,Y 253.17,Z 369.545,A -85,B 0,C 180,E1 -21093.185,E2 -21093.185} C_VEL
LIN {X 0,Y 250.169,Z 414.595,A -85,B 0,C 180,E1 -21094.416,E2 -21094.416} C_VEL
LIN {X 0,Y 248.38,Z 428.363,A -85,B 0,C 180,E1 -21095.038,E2 -21095.038} C_VEL
LIN {X 0,Y 245.795,Z 442.212,A -85,B 0,C 180,E1 -21095.952,E2 -21095.952} C_VEL
LIN {X 0,Y 243.097,Z 453.748,A -85,B 0,C 180,E1 -21096.98,E2 -21096.98} C_VEL
LIN {X 0,Y 239.72,Z 465.717,A -85,B 0,C 180,E1 -21098.351,E2 -21098.351} C_VEL
LIN {X 0,Y 235.591,Z 477.999,A -85,B 0,C 180,E1 -21100.146,E2 -21100.146} C_VEL
LIN {X 0,Y 230.968,Z 489.583,A -85,B 0,C 180,E1 -21102.276,E2 -21102.276} C_VEL
LIN {X 0,Y 226.65,Z 499.195,A -85,B 0,C 180,E1 -21104.507,E2 -21104.507} C_VEL
LIN {X 0,Y 222.264,Z 508.285,A -85,B 0,C 180,E1 -21107.171,E2 -21107.171} C_VEL
LIN {X 0,Y 218.283,Z 515.754,A -85,B 0,C 180,E1 -21109.915,E2 -21109.915} C_VEL
LIN {X 0,Y 214.874,Z 521.893,A -85,B 0,C 180,E1 -21112.766,E2 -21112.766} C_VEL
LIN {X 0,Y 211.53,Z 527.586,A -85,B 0,C 180,E1 -21116.156,E2 -21116.156} C_VEL
LIN {X 0,Y 208.805,Z 531.972,A -85,B 0,C 180,E1 -21119.678,E2 -21119.678} C_VEL
LIN {X 0,Y 206.543,Z 535.431,A -85,B 0,C 180,E1 -21123.747,E2 -21123.747} C_VEL
LIN {X 0,Y 205.084,Z 537.356,A -85,B 0,C 180,E1 -21127.855,E2 -21127.855} C_VEL
LIN {X 0,Y 204.293,Z 537.837,A -85,B 0,C 180,E1 -21131.965,E2 -21131.965} C_VEL
LIN {X 0,Y 204.043,Z 536.923,A -85,B 0,C 180,E1 -21136.049,E2 -21136.049} C_VEL
LIN {X 0,Y 204.156,Z 534.629,A -85,B 0,C 180,E1 -21140.089,E2 -21140.089} C_VEL
LIN {X 0,Y 204.868,Z 530.849,A -85,B 0,C 180,E1 -21144.147,E2 -21144.147} C_VEL
LIN {X 0,Y 205.789,Z 525.692,A -85,B 0,C 180,E1 -21148.043,E2 -21148.043} C_VEL
LIN {X 0,Y 206.902,Z 520.632,A -85,B 0,C 180,E1 -21150.973,E2 -21150.973} C_VEL
LIN {X 0,Y 208.774,Z 513.4,A -85,B 0,C 180,E1 -21154.344,E2 -21154.344} C_VEL
LIN {X 0,Y 210.795,Z 505.832,A -85,B 0,C 180,E1 -21157.182,E2 -21157.182} C_VEL
LIN {X 0,Y 213.29,Z 496.74,A -85,B 0,C 180,E1 -21159.962,E2 -21159.962} C_VEL
LIN {X 0,Y 216.157,Z 485.927,A -85,B 0,C 180,E1 -21162.63,E2 -21162.63} C_VEL
LIN {X 0,Y 218.892,Z 474.519,A -85,B 0,C 180,E1 -21164.884,E2 -21164.884} C_VEL
LIN {X 0,Y 221.386,Z 462.174,A -85,B 0,C 180,E1 -21166.838,E2 -21166.838} C_VEL
LIN {X 0,Y 223.793,Z 450.185,A -85,B 0,C 180,E1 -21168.303,E2 -21168.303} C_VEL
LIN {X 0,Y 225.696,Z 437.187,A -85,B 0,C 180,E1 -21169.557,E2 -21169.557} C_VEL
LIN {X 0,Y 227.231,Z 423.229,A -85,B 0,C 180,E1 -21170.539,E2 -21170.539} C_VEL
LIN {X 0,Y 228.338,Z 408.593,A -85,B 0,C 180,E1 -21171.201,E2 -21171.201} C_VEL
LIN {X 0,Y 231.915,Z 332.816,A -85,B 0,C 180,E1 -21173.423,E2 -21173.423} C_VEL
LIN {X 0,Y 224.63,Z 314.186,A -85,B 0,C 180,E1 -21175.313,E2 -21175.313} C_VEL
LIN {X 0,Y 215.299,Z 297.055,A -85,B 0,C 180,E1 -21177.701,E2 -21177.701} C_VEL
LIN {X 0,Y 210.402,Z 289.241,A -85,B 0,C 180,E1 -21179.02,E2 -21179.02} C_VEL
LIN {X 0,Y 208.747,Z 286.484,A -85,B 0,C 180,E1 -21179.491,E2 -21179.491} C_VEL
LIN {X 0,Y 207.114,Z 283.976,A -85,B 0,C 180,E1 -21179.956,E2 -21179.956} C_VEL
LIN {X 0,Y 206.711,Z 282.348,A -85,B 0,C 180,E1 -21180.124,E2 -21180.124} C_VEL
LIN {X 0,Y 206.712,Z 282.36,A -85,B 0,C 180,E1 -21185.322,E2 -21185.322} C_VEL
LIN {X 0,Y 206.751,Z 282.355,A -85,B 0,C 180,E1 -21188.577,E2 -21188.577} C_VEL
LIN {X 0,Y 206.728,Z 282.357,A -85,B 0,C 180,E1 -21192.837,E2 -21192.837} C_VEL
LIN {X 0,Y 206.735,Z 282.339,A -85,B 0,C 180,E1 -21197.168,E2 -21197.168} C_VEL
LIN {X 0,Y 206.753,Z 282.35,A -85,B 0,C 180,E1 -21201.426,E2 -21201.426} C_VEL
LIN {X 0,Y 206.723,Z 282.334,A -85,B 0,C 180,E1 -21204.697,E2 -21204.697} C_VEL
LIN {X 0,Y 206.716,Z 282.357,A -85,B 0,C 180,E1 -21209.341,E2 -21209.341} C_VEL
LIN {X 0,Y 206.725,Z 282.334,A -85,B 0,C 180,E1 -21213.774,E2 -21213.774} C_VEL
LIN {X 0,Y 206.751,Z 282.356,A -85,B 0,C 180,E1 -21218.046,E2 -21218.046} C_VEL
LIN {X 0,Y 206.867,Z 282.34,A -85,B 0,C 180,E1 -21222.199,E2 -21222.199} C_VEL
LIN {X 0,Y 206.888,Z 282.333,A -85,B 0,C 180,E1 -21226.247,E2 -21226.247} C_VEL
LIN {X 0,Y 207.095,Z 282.304,A -85,B 0,C 180,E1 -21230.234,E2 -21230.234} C_VEL
LIN {X 0,Y 207.057,Z 282.293,A -85,B 0,C 180,E1 -21234.158,E2 -21234.158} C_VEL
LIN {X 0,Y 207.378,Z 282.277,A -85,B 0,C 180,E1 -21238.061,E2 -21238.061} C_VEL
LIN {X 0,Y 207.511,Z 282.255,A -85,B 0,C 180,E1 -21240.003,E2 -21240.003} C_VEL
LIN {X 0,Y 207.378,Z 282.254,A -85,B 0,C 180,E1 -21241.945,E2 -21241.945} C_VEL
LIN {X 0,Y 207.138,Z 282.308,A -85,B 0,C 180,E1 -21247.803,E2 -21247.803} C_VEL
LIN {X 0,Y 206.922,Z 282.312,A -85,B 0,C 180,E1 -21251.761,E2 -21251.761} C_VEL
LIN {X 0,Y 206.863,Z 282.339,A -85,B 0,C 180,E1 -21255.774,E2 -21255.774} C_VEL
LIN {X 0,Y 206.762,Z 282.349,A -85,B 0,C 180,E1 -21259.874,E2 -21259.874} C_VEL
LIN {X 0,Y 206.748,Z 282.352,A -85,B 0,C 180,E1 -21264.077,E2 -21264.077} C_VEL
LIN {X 0,Y 206.746,Z 282.356,A -85,B 0,C 180,E1 -21268.421,E2 -21268.421} C_VEL
LIN {X 0,Y 206.701,Z 282.363,A -85,B 0,C 180,E1 -21272.96,E2 -21272.96} C_VEL
LIN {X 0,Y 206.683,Z 282.362,A -85,B 0,C 180,E1 -21277.742,E2 -21277.742} C_VEL
LIN {X 0,Y 206.645,Z 282.371,A -85,B 0,C 180,E1 -21281.565,E2 -21281.565} C_VEL
LIN {X 0,Y 206.626,Z 282.369,A -85,B 0,C 180,E1 -21282.833,E2 -21282.833} C_VEL
LIN {X 0,Y 206.722,Z 283.086,A -85,B 0,C 180,E1 -21283.703,E2 -21283.703} C_VEL
LIN {X 0,Y 207.01,Z 285.451,A -85,B 0,C 180,E1 -21284.665,E2 -21284.665} C_VEL
LIN {X 0,Y 207.392,Z 288.424,A -85,B 0,C 180,E1 -21285.37,E2 -21285.37} C_VEL
LIN {X 0,Y 207.88,Z 291.796,A -85,B 0,C 180,E1 -21285.918,E2 -21285.918} C_VEL
LIN {X 0,Y 209.383,Z 299.9,A -85,B 0,C 180,E1 -21286.829,E2 -21286.829} C_VEL
LIN {X 0,Y 211.17,Z 305.855,A -85,B 0,C 180,E1 -21287.465,E2 -21287.465} C_VEL
LIN {X 0,Y 211.956,Z 307.73,A -85,B 0,C 180,E1 -21287.702,E2 -21287.702} C_VEL
LIN {X 0,Y 218.516,Z 322.732,A -85,B 0,C 180,E1 -21289.566,E2 -21289.566} C_VEL
LIN {X 0,Y 224.248,Z 338.081,A -85,B 0,C 180,E1 -21291.162,E2 -21291.162} C_VEL
LIN {X 0,Y 225.406,Z 347.857,A -85,B 0,C 180,E1 -21291.722,E2 -21291.722} C_VEL
LIN {X 0,Y 221.791,Z 423.705,A -85,B 0,C 180,E1 -21294.042,E2 -21294.042} C_VEL
LIN {X 0,Y 220.476,Z 437.727,A -85,B 0,C 180,E1 -21294.777,E2 -21294.777} C_VEL
LIN {X 0,Y 218.36,Z 451.966,A -85,B 0,C 180,E1 -21295.86,E2 -21295.86} C_VEL
LIN {X 0,Y 215.917,Z 465.161,A -85,B 0,C 180,E1 -21297.24,E2 -21297.24} C_VEL
LIN {X 0,Y 213.294,Z 477.902,A -85,B 0,C 180,E1 -21299.003,E2 -21299.003} C_VEL
LIN {X 0,Y 211.088,Z 487.214,A -85,B 0,C 180,E1 -21300.588,E2 -21300.588} C_VEL
LIN {X 0,Y 208.294,Z 498.288,A -85,B 0,C 180,E1 -21302.903,E2 -21302.903} C_VEL
LIN {X 0,Y 205.664,Z 507.524,A -85,B 0,C 180,E1 -21305.253,E2 -21305.253} C_VEL
LIN {X 0,Y 203.09,Z 516.788,A -85,B 0,C 180,E1 -21308.161,E2 -21308.161} C_VEL
LIN {X 0,Y 201.13,Z 523.835,A -85,B 0,C 180,E1 -21310.842,E2 -21310.842} C_VEL
LIN {X 0,Y 199.76,Z 529.896,A -85,B 0,C 180,E1 -21313.653,E2 -21313.653} C_VEL
LIN {X 0,Y 198.502,Z 535.321,A -85,B 0,C 180,E1 -21316.695,E2 -21316.695} C_VEL
LIN {X 0,Y 197.623,Z 541.018,A -85,B 0,C 180,E1 -21320.791,E2 -21320.791} C_VEL
LIN {X 0,Y 197.31,Z 544.203,A -85,B 0,C 180,E1 -21323.866,E2 -21323.866} C_VEL
LIN {X 0,Y 197.275,Z 547.155,A -85,B 0,C 180,E1 -21327.958,E2 -21327.958} C_VEL
LIN {X 0,Y 197.401,Z 548.103,A -85,B 0,C 180,E1 -21330,E2 -21330} C_VEL
LIN {X 0,Y 197.212,Z 548.96,A -85,B 0,C 180,E1 -21334.087,E2 -21334.087} C_VEL
LIN {X 0,Y 197.502,Z 548.499,A -85,B 0,C 180,E1 -21338.183,E2 -21338.183} C_VEL
LIN {X 0,Y 198.457,Z 546.731,A -85,B 0,C 180,E1 -21342.267,E2 -21342.267} C_VEL
LIN {X 0,Y 200.263,Z 543.626,A -85,B 0,C 180,E1 -21346.304,E2 -21346.304} C_VEL
LIN {X 0,Y 202.946,Z 539.103,A -85,B 0,C 180,E1 -21350.26,E2 -21350.26} C_VEL
LIN {X 0,Y 205.528,Z 534.654,A -85,B 0,C 180,E1 -21353.155,E2 -21353.155} C_VEL
LIN {X 0,Y 209.852,Z 527.269,A -85,B 0,C 180,E1 -21356.879,E2 -21356.879} C_VEL
LIN {X 0,Y 214.416,Z 519.144,A -85,B 0,C 180,E1 -21359.989,E2 -21359.989} C_VEL
LIN {X 0,Y 218.851,Z 510.679,A -85,B 0,C 180,E1 -21362.539,E2 -21362.539} C_VEL
LIN {X 0,Y 223.531,Z 500.831,A -85,B 0,C 180,E1 -21364.913,E2 -21364.913} C_VEL
LIN {X 0,Y 227.932,Z 490.28,A -85,B 0,C 180,E1 -21366.959,E2 -21366.959} C_VEL
LIN {X 0,Y 232.661,Z 477.819,A -85,B 0,C 180,E1 -21368.813,E2 -21368.813} C_VEL
LIN {X 0,Y 236.018,Z 467.261,A -85,B 0,C 180,E1 -21370.085,E2 -21370.085} C_VEL
LIN {X 0,Y 239.669,Z 454.005,A -85,B 0,C 180,E1 -21371.282,E2 -21371.282} C_VEL
LIN {X 0,Y 242.519,Z 440.306,A -85,B 0,C 180,E1 -21372.217,E2 -21372.217} C_VEL
LIN {X 0,Y 244.647,Z 426.112,A -85,B 0,C 180,E1 -21372.879,E2 -21372.879} C_VEL
LIN {X 0,Y 246.139,Z 407.718,A -85,B 0,C 180,E1 -21373.427,E2 -21373.427} C_VEL
LIN {X 0,Y 249.125,Z 361.78,A -85,B 0,C 180,E1 -21374.656,E2 -21374.656} C_VEL
LIN {X 0,Y 244.876,Z 351.703,A -85,B 0,C 180,E1 -21376.336,E2 -21376.336} C_VEL
LIN {X 0,Y 239.556,Z 340.806,A -85,B 0,C 180,E1 -21378.54,E2 -21378.54} C_VEL
LIN {X 0,Y 234.973,Z 332.333,A -85,B 0,C 180,E1 -21380.584,E2 -21380.584} C_VEL
LIN {X 0,Y 229.745,Z 323.466,A -85,B 0,C 180,E1 -21383.135,E2 -21383.135} C_VEL
LIN {X 0,Y 226.899,Z 318.894,A -85,B 0,C 180,E1 -21384.643,E2 -21384.643} C_VEL
LIN {X 0,Y 223.377,Z 313.557,A -85,B 0,C 180,E1 -21386.647,E2 -21386.647} C_VEL
LIN {X 0,Y 219.709,Z 308.228,A -85,B 0,C 180,E1 -21388.948,E2 -21388.948} C_VEL
LIN {X 0,Y 216.282,Z 303.29,A -85,B 0,C 180,E1 -21391.4,E2 -21391.4} C_VEL
LIN {X 0,Y 211.034,Z 296.421,A -85,B 0,C 180,E1 -21395.905,E2 -21395.905} C_VEL
LIN {X 0,Y 209.525,Z 294.78,A -85,B 0,C 180,E1 -21397.429,E2 -21397.429} C_VEL
LIN {X 0,Y 206.958,Z 292.647,A -85,B 0,C 180,E1 -21400.404,E2 -21400.404} C_VEL
LIN {X 0,Y 205.745,Z 290.05,A -85,B 0,C 180,E1 -21402.383,E2 -21402.383} C_VEL
LIN {X 0,Y 205.543,Z 289.314,A -85,B 0,C 180,E1 -21402.806,E2 -21402.806} C_VEL
LIN {X 0,Y 202.338,Z 287.517,A -85,B 0,C 180,E1 -21412.011,E2 -21412.011} C_VEL
LIN {X 0,Y 203.682,Z 288.217,A -85,B 0,C 180,E1 -21419.997,E2 -21419.997} C_VEL
LIN {X 0,Y 205.806,Z 289.501,A -85,B 0,C 180,E1 -21424.036,E2 -21424.036} C_VEL
LIN {X 0,Y 206.971,Z 292.156,A -85,B 0,C 180,E1 -21425.966,E2 -21425.966} C_VEL
LIN {X 0,Y 209.712,Z 294.664,A -85,B 0,C 180,E1 -21429.157,E2 -21429.157} C_VEL
LIN {X 0,Y 210.79,Z 295.413,A -85,B 0,C 180,E1 -21430.202,E2 -21430.202} C_VEL
LIN {X 0,Y 212.333,Z 298.285,A -85,B 0,C 180,E1 -21431.77,E2 -21431.77} C_VEL
LIN {X 0,Y 214.898,Z 300.565,A -85,B 0,C 180,E1 -21433.864,E2 -21433.864} C_VEL
LIN {X 0,Y 215.763,Z 301.823,A -85,B 0,C 180,E1 -21434.559,E2 -21434.559} C_VEL
LIN {X 0,Y 218.324,Z 305.14,A -85,B 0,C 180,E1 -21436.44,E2 -21436.44} C_VEL
LIN {X 0,Y 219.589,Z 306.482,A -85,B 0,C 180,E1 -21437.278,E2 -21437.278} C_VEL
LIN {X 0,Y 222.437,Z 310.229,A -85,B 0,C 180,E1 -21439.077,E2 -21439.077} C_VEL
LIN {X 0,Y 223.811,Z 311.997,A -85,B 0,C 180,E1 -21439.886,E2 -21439.886} C_VEL
LIN {X 0,Y 227.41,Z 316.715,A -85,B 0,C 180,E1 -21441.874,E2 -21441.874} C_VEL
LIN {X 0,Y 231.625,Z 322.585,A -85,B 0,C 180,E1 -21444.007,E2 -21444.007} C_VEL
LIN {X 0,Y 236.98,Z 330.506,A -85,B 0,C 180,E1 -21446.47,E2 -21446.47} C_VEL
LIN {X 0,Y 241.841,Z 338.879,A -85,B 0,C 180,E1 -21448.535,E2 -21448.535} C_VEL
LIN {X 0,Y 248.092,Z 351.253,A -85,B 0,C 180,E1 -21451.009,E2 -21451.009} C_VEL
LIN {X 0,Y 249.515,Z 354.363,A -85,B 0,C 180,E1 -21451.55,E2 -21451.55} C_VEL
LIN {X 0,Y 245.435,Z 414.46,A -85,B 0,C 180,E1 -21453.187,E2 -21453.187} C_VEL
LIN {X 0,Y 243.515,Z 428.778,A -85,B 0,C 180,E1 -21453.837,E2 -21453.837} C_VEL
LIN {X 0,Y 240.988,Z 441.989,A -85,B 0,C 180,E1 -21454.713,E2 -21454.713} C_VEL
LIN {X 0,Y 237.866,Z 454.746,A -85,B 0,C 180,E1 -21455.86,E2 -21455.86} C_VEL
LIN {X 0,Y 234.189,Z 467.135,A -85,B 0,C 180,E1 -21457.322,E2 -21457.322} C_VEL
LIN {X 0,Y 229.914,Z 479.198,A -85,B 0,C 180,E1 -21459.137,E2 -21459.137} C_VEL
LIN {X 0,Y 225.456,Z 489.873,A -85,B 0,C 180,E1 -21461.145,E2 -21461.145} C_VEL
LIN {X 0,Y 220.662,Z 500.086,A -85,B 0,C 180,E1 -21463.568,E2 -21463.568} C_VEL
LIN {X 0,Y 216.021,Z 509.207,A -85,B 0,C 180,E1 -21466.336,E2 -21466.336} C_VEL
LIN {X 0,Y 211.448,Z 517.297,A -85,B 0,C 180,E1 -21469.478,E2 -21469.478} C_VEL
LIN {X 0,Y 207.814,Z 523.381,A -85,B 0,C 180,E1 -21472.503,E2 -21472.503} C_VEL
LIN {X 0,Y 204.95,Z 527.912,A -85,B 0,C 180,E1 -21475.38,E2 -21475.38} C_VEL
LIN {X 0,Y 202.34,Z 531.84,A -85,B 0,C 180,E1 -21478.601,E2 -21478.601} C_VEL
LIN {X 0,Y 200.833,Z 534.104,A -85,B 0,C 180,E1 -21481.021,E2 -21481.021} C_VEL
LIN {X 0,Y 198.925,Z 536.621,A -85,B 0,C 180,E1 -21484.916,E2 -21484.916} C_VEL
LIN {X 0,Y 197.644,Z 537.949,A -85,B 0,C 180,E1 -21489.171,E2 -21489.171} C_VEL
LIN {X 0,Y 197.051,Z 537.833,A -85,B 0,C 180,E1 -21493.422,E2 -21493.422} C_VEL
LIN {X 0,Y 196.974,Z 537.251,A -85,B 0,C 180,E1 -21495.537,E2 -21495.537} C_VEL
LIN {X 0,Y 197.038,Z 535.054,A -85,B 0,C 180,E1 -21499.727,E2 -21499.727} C_VEL
LIN {X 0,Y 197.702,Z 531.434,A -85,B 0,C 180,E1 -21503.878,E2 -21503.878} C_VEL
LIN {X 0,Y 198.362,Z 527.76,A -85,B 0,C 180,E1 -21506.954,E2 -21506.954} C_VEL
LIN {X 0,Y 199.394,Z 523.157,A -85,B 0,C 180,E1 -21510,E2 -21510} C_VEL
LIN {X 0,Y 201.067,Z 516.499,A -85,B 0,C 180,E1 -21513.507,E2 -21513.507} C_VEL
LIN {X 0,Y 203.364,Z 508.207,A -85,B 0,C 180,E1 -21516.947,E2 -21516.947} C_VEL
LIN {X 0,Y 205.845,Z 499.551,A -85,B 0,C 180,E1 -21519.829,E2 -21519.829} C_VEL
LIN {X 0,Y 208.854,Z 488.673,A -85,B 0,C 180,E1 -21522.733,E2 -21522.733} C_VEL
LIN {X 0,Y 211.795,Z 477.314,A -85,B 0,C 180,E1 -21525.151,E2 -21525.151} C_VEL
LIN {X 0,Y 214.432,Z 465.602,A -85,B 0,C 180,E1 -21527.156,E2 -21527.156} C_VEL
LIN {X 0,Y 216.676,Z 454.43,A -85,B 0,C 180,E1 -21528.681,E2 -21528.681} C_VEL
LIN {X 0,Y 218.897,Z 441.432,A -85,B 0,C 180,E1 -21530.068,E2 -21530.068} C_VEL
LIN {X 0,Y 220.65,Z 427.511,A -85,B 0,C 180,E1 -21531.181,E2 -21531.181} C_VEL
LIN {X 0,Y 221.994,Z 412.878,A -85,B 0,C 180,E1 -21531.96,E2 -21531.96} C_VEL
LIN {X 0,Y 225.965,Z 334.906,A -85,B 0,C 180,E1 -21534.301,E2 -21534.301} C_VEL
LIN {X 0,Y 219.359,Z 317.895,A -85,B 0,C 180,E1 -21536.098,E2 -21536.098} C_VEL
LIN {X 0,Y 210.295,Z 301.132,A -85,B 0,C 180,E1 -21538.536,E2 -21538.536} C_VEL
LIN {X 0,Y 203.922,Z 290.907,A -85,B 0,C 180,E1 -21540.362,E2 -21540.362} C_VEL
LIN {X 0,Y 201.671,Z 287.345,A -85,B 0,C 180,E1 -21541.04,E2 -21541.04} C_VEL
LIN {X 0,Y 200.15,Z 285.056,A -85,B 0,C 180,E1 -21541.505,E2 -21541.505} C_VEL
LIN {X 0,Y 199.676,Z 283.237,A -85,B 0,C 180,E1 -21541.756,E2 -21541.756} C_VEL
LIN {X 0,Y 199.644,Z 283.239,A -85,B 0,C 180,E1 -21546.758,E2 -21546.758} C_VEL
LIN {X 0,Y 199.669,Z 283.228,A -85,B 0,C 180,E1 -21549.313,E2 -21549.313} C_VEL
LIN {X 0,Y 199.67,Z 283.236,A -85,B 0,C 180,E1 -21552.345,E2 -21552.345} C_VEL
LIN {X 0,Y 199.685,Z 283.224,A -85,B 0,C 180,E1 -21555.263,E2 -21555.263} C_VEL
LIN {X 0,Y 199.684,Z 283.222,A -85,B 0,C 180,E1 -21558.036,E2 -21558.036} C_VEL
LIN {X 0,Y 199.694,Z 283.234,A -85,B 0,C 180,E1 -21560.737,E2 -21560.737} C_VEL
LIN {X 0,Y 199.626,Z 283.224,A -85,B 0,C 180,E1 -21565.72,E2 -21565.72} C_VEL
LIN {X 0,Y 199.696,Z 283.232,A -85,B 0,C 180,E1 -21568.14,E2 -21568.14} C_VEL
LIN {X 0,Y 199.679,Z 283.208,A -85,B 0,C 180,E1 -21572.774,E2 -21572.774} C_VEL
LIN {X 0,Y 199.731,Z 283.231,A -85,B 0,C 180,E1 -21577.232,E2 -21577.232} C_VEL
LIN {X 0,Y 199.791,Z 283.221,A -85,B 0,C 180,E1 -21581.76,E2 -21581.76} C_VEL
LIN {X 0,Y 199.83,Z 283.211,A -85,B 0,C 180,E1 -21585.751,E2 -21585.751} C_VEL
LIN {X 0,Y 200.018,Z 283.189,A -85,B 0,C 180,E1 -21589.884,E2 -21589.884} C_VEL
LIN {X 0,Y 200.018,Z 283.167,A -85,B 0,C 180,E1 -21593.952,E2 -21593.952} C_VEL
LIN {X 0,Y 200.317,Z 283.157,A -85,B 0,C 180,E1 -21597.992,E2 -21597.992} C_VEL
LIN {X 0,Y 200.476,Z 283.13,A -85,B 0,C 180,E1 -21600.003,E2 -21600.003} C_VEL
LIN {X 0,Y 200.022,Z 283.169,A -85,B 0,C 180,E1 -21604.032,E2 -21604.032} C_VEL
LIN {X 0,Y 200.087,Z 283.187,A -85,B 0,C 180,E1 -21608.079,E2 -21608.079} C_VEL
LIN {X 0,Y 199.872,Z 283.187,A -85,B 0,C 180,E1 -21612.182,E2 -21612.182} C_VEL
LIN {X 0,Y 199.802,Z 283.222,A -85,B 0,C 180,E1 -21616.346,E2 -21616.346} C_VEL
LIN {X 0,Y 199.681,Z 283.237,A -85,B 0,C 180,E1 -21620.61,E2 -21620.61} C_VEL
LIN {X 0,Y 199.666,Z 283.238,A -85,B 0,C 180,E1 -21624.988,E2 -21624.988} C_VEL
LIN {X 0,Y 199.672,Z 283.239,A -85,B 0,C 180,E1 -21629.525,E2 -21629.525} C_VEL
LIN {X 0,Y 199.674,Z 283.239,A -85,B 0,C 180,E1 -21632.358,E2 -21632.358} C_VEL
LIN {X 0,Y 199.626,Z 283.244,A -85,B 0,C 180,E1 -21636.765,E2 -21636.765} C_VEL
LIN {X 0,Y 199.612,Z 283.247,A -85,B 0,C 180,E1 -21639.33,E2 -21639.33} C_VEL
LIN {X 0,Y 199.629,Z 283.324,A -85,B 0,C 180,E1 -21643.106,E2 -21643.106} C_VEL
LIN {X 0,Y 200.258,Z 285.413,A -85,B 0,C 180,E1 -21644.167,E2 -21644.167} C_VEL
LIN {X 0,Y 202.707,Z 289.854,A -85,B 0,C 180,E1 -21644.945,E2 -21644.945} C_VEL
LIN {X 0,Y 210.38,Z 304.593,A -85,B 0,C 180,E1 -21647.252,E2 -21647.252} C_VEL
LIN {X 0,Y 211.956,Z 307.73,A -85,B 0,C 180,E1 -21647.702,E2 -21647.702} C_VEL
LIN {X 0,Y 213.623,Z 313.038,A -85,B 0,C 180,E1 -21648.252,E2 -21648.252} C_VEL
LIN {X 0,Y 214.717,Z 322.701,A -85,B 0,C 180,E1 -21648.858,E2 -21648.858} C_VEL
LIN {X 0,Y 215.816,Z 332.375,A -85,B 0,C 180,E1 -21649.456,E2 -21649.456} C_VEL
LIN {X 0,Y 217.517,Z 337.701,A -85,B 0,C 180,E1 -21649.979,E2 -21649.979} C_VEL
LIN {X 0,Y 218.587,Z 341.3,A -85,B 0,C 180,E1 -21650.313,E2 -21650.313} C_VEL
LIN {X 0,Y 219.409,Z 349.309,A -85,B 0,C 180,E1 -21650.77,E2 -21650.77} C_VEL
LIN {X 0,Y 215.724,Z 423.471,A -85,B 0,C 180,E1 -21653.083,E2 -21653.083} C_VEL
LIN {X 0,Y 214.347,Z 437.5,A -85,B 0,C 180,E1 -21653.831,E2 -21653.831} C_VEL
LIN {X 0,Y 212.287,Z 451.184,A -85,B 0,C 180,E1 -21654.886,E2 -21654.886} C_VEL
LIN {X 0,Y 209.928,Z 463.609,A -85,B 0,C 180,E1 -21656.181,E2 -21656.181} C_VEL
LIN {X 0,Y 207.33,Z 475.862,A -85,B 0,C 180,E1 -21657.86,E2 -21657.86} C_VEL
LIN {X 0,Y 204.935,Z 486.125,A -85,B 0,C 180,E1 -21659.614,E2 -21659.614} C_VEL
LIN {X 0,Y 202.48,Z 495.253,A -85,B 0,C 180,E1 -21661.494,E2 -21661.494} C_VEL
LIN {X 0,Y 199.646,Z 504.92,A -85,B 0,C 180,E1 -21663.895,E2 -21663.895} C_VEL
LIN {X 0,Y 196.867,Z 514.624,A -85,B 0,C 180,E1 -21666.878,E2 -21666.878} C_VEL
LIN {X 0,Y 194.646,Z 522.448,A -85,B 0,C 180,E1 -21669.852,E2 -21669.852} C_VEL
LIN {X 0,Y 192.872,Z 529.307,A -85,B 0,C 180,E1 -21673.052,E2 -21673.052} C_VEL
LIN {X 0,Y 191.558,Z 534.813,A -85,B 0,C 180,E1 -21676.203,E2 -21676.203} C_VEL
LIN {X 0,Y 190.562,Z 540.58,A -85,B 0,C 180,E1 -21680.447,E2 -21680.447} C_VEL
LIN {X 0,Y 190.23,Z 543.833,A -85,B 0,C 180,E1 -21683.636,E2 -21683.636} C_VEL
LIN {X 0,Y 190.183,Z 546.849,A -85,B 0,C 180,E1 -21687.882,E2 -21687.882} C_VEL
LIN {X 0,Y 190.302,Z 547.827,A -85,B 0,C 180,E1 -21690,E2 -21690} C_VEL
LIN {X 0,Y 190.133,Z 548.745,A -85,B 0,C 180,E1 -21694.239,E2 -21694.239} C_VEL
LIN {X 0,Y 190.462,Z 548.343,A -85,B 0,C 180,E1 -21698.487,E2 -21698.487} C_VEL
LIN {X 0,Y 191.48,Z 546.636,A -85,B 0,C 180,E1 -21702.721,E2 -21702.721} C_VEL
LIN {X 0,Y 193.428,Z 543.595,A -85,B 0,C 180,E1 -21706.897,E2 -21706.897} C_VEL
LIN {X 0,Y 196.246,Z 539.142,A -85,B 0,C 180,E1 -21710.984,E2 -21710.984} C_VEL
LIN {X 0,Y 200.045,Z 533.142,A -85,B 0,C 180,E1 -21714.934,E2 -21714.934} C_VEL
LIN {X 0,Y 204.189,Z 526.436,A -85,B 0,C 180,E1 -21718.245,E2 -21718.245} C_VEL
LIN {X 0,Y 209.022,Z 518.131,A -85,B 0,C 180,E1 -21721.409,E2 -21721.409} C_VEL
LIN {X 0,Y 213.729,Z 509.51,A -85,B 0,C 180,E1 -21723.986,E2 -21723.986} C_VEL
LIN {X 0,Y 218.865,Z 498.793,A -85,B 0,C 180,E1 -21726.538,E2 -21726.538} C_VEL
LIN {X 0,Y 223.291,Z 488.665,A -85,B 0,C 180,E1 -21728.434,E2 -21728.434} C_VEL
LIN {X 0,Y 227.698,Z 477.317,A -85,B 0,C 180,E1 -21730.113,E2 -21730.113} C_VEL
LIN {X 0,Y 231.755,Z 464.926,A -85,B 0,C 180,E1 -21731.555,E2 -21731.555} C_VEL
LIN {X 0,Y 235.487,Z 451.099,A -85,B 0,C 180,E1 -21732.761,E2 -21732.761} C_VEL
LIN {X 0,Y 238.199,Z 437.967,A -85,B 0,C 180,E1 -21733.603,E2 -21733.603} C_VEL
LIN {X 0,Y 240.275,Z 423.847,A -85,B 0,C 180,E1 -21734.219,E2 -21734.219} C_VEL
LIN {X 0,Y 243.443,Z 379.178,A -85,B 0,C 180,E1 -21735.469,E2 -21735.469} C_VEL
LIN {X 0,Y 244.397,Z 364.035,A -85,B 0,C 180,E1 -21735.898,E2 -21735.898} C_VEL
LIN {X 0,Y 239.822,Z 353.45,A -85,B 0,C 180,E1 -21737.817,E2 -21737.817} C_VEL
LIN {X 0,Y 234.602,Z 342.661,A -85,B 0,C 180,E1 -21740.154,E2 -21740.154} C_VEL
LIN {X 0,Y 229.755,Z 333.881,A -85,B 0,C 180,E1 -21742.508,E2 -21742.508} C_VEL
LIN {X 0,Y 224.955,Z 325.631,A -85,B 0,C 180,E1 -21745.088,E2 -21745.088} C_VEL
LIN {X 0,Y 220.845,Z 319.349,A -85,B 0,C 180,E1 -21747.519,E2 -21747.519} C_VEL
LIN {X 0,Y 217.558,Z 314.398,A -85,B 0,C 180,E1 -21749.695,E2 -21749.695} C_VEL
LIN {X 0,Y 213.752,Z 308.888,A -85,B 0,C 180,E1 -21752.59,E2 -21752.59} C_VEL
LIN {X 0,Y 208.833,Z 302.157,A -85,B 0,C 180,E1 -21757.189,E2 -21757.189} C_VEL
LIN {X 0,Y 205.543,Z 299.181,A -85,B 0,C 180,E1 -21761.107,E2 -21761.107} C_VEL
LIN {X 0,Y 204.397,Z 296.363,A -85,B 0,C 180,E1 -21763.197,E2 -21763.197} C_VEL
LIN {X 0,Y 201.464,Z 294.564,A -85,B 0,C 180,E1 -21771.976,E2 -21771.976} C_VEL
LIN {X 0,Y 202.801,Z 295.276,A -85,B 0,C 180,E1 -21779.997,E2 -21779.997} C_VEL
LIN {X 0,Y 204.612,Z 296.424,A -85,B 0,C 180,E1 -21783.567,E2 -21783.567} C_VEL
LIN {X 0,Y 205.88,Z 299.18,A -85,B 0,C 180,E1 -21785.737,E2 -21785.737} C_VEL
LIN {X 0,Y 208.838,Z 301.765,A -85,B 0,C 180,E1 -21789.195,E2 -21789.195} C_VEL
LIN {X 0,Y 209.335,Z 302.344,A -85,B 0,C 180,E1 -21789.715,E2 -21789.715} C_VEL
LIN {X 0,Y 211.316,Z 305.572,A -85,B 0,C 180,E1 -21791.721,E2 -21791.721} C_VEL
LIN {X 0,Y 213.679,Z 307.756,A -85,B 0,C 180,E1 -21793.679,E2 -21793.679} C_VEL
LIN {X 0,Y 216.1,Z 311.232,A -85,B 0,C 180,E1 -21795.585,E2 -21795.585} C_VEL
LIN {X 0,Y 217.665,Z 312.981,A -85,B 0,C 180,E1 -21796.681,E2 -21796.681} C_VEL
LIN {X 0,Y 220.67,Z 316.907,A -85,B 0,C 180,E1 -21798.642,E2 -21798.642} C_VEL
LIN {X 0,Y 225.103,Z 322.995,A -85,B 0,C 180,E1 -21801.236,E2 -21801.236} C_VEL
LIN {X 0,Y 229.981,Z 329.848,A -85,B 0,C 180,E1 -21803.772,E2 -21803.772} C_VEL
LIN {X 0,Y 235.383,Z 338.405,A -85,B 0,C 180,E1 -21806.324,E2 -21806.324} C_VEL
LIN {X 0,Y 240.774,Z 348.546,A -85,B 0,C 180,E1 -21808.673,E2 -21808.673} C_VEL
LIN {X 0,Y 244.906,Z 357.212,A -85,B 0,C 180,E1 -21810.36,E2 -21810.36} C_VEL
LIN {X 0,Y 240.823,Z 414.441,A -85,B 0,C 180,E1 -21811.915,E2 -21811.915} C_VEL
LIN {X 0,Y 238.764,Z 429.231,A -85,B 0,C 180,E1 -21812.589,E2 -21812.589} C_VEL
LIN {X 0,Y 236.021,Z 442.958,A -85,B 0,C 180,E1 -21813.516,E2 -21813.516} C_VEL
LIN {X 0,Y 232.824,Z 455.44,A -85,B 0,C 180,E1 -21814.66,E2 -21814.66} C_VEL
LIN {X 0,Y 229.037,Z 467.632,A -85,B 0,C 180,E1 -21816.117,E2 -21816.117} C_VEL
LIN {X 0,Y 224.788,Z 479.171,A -85,B 0,C 180,E1 -21817.869,E2 -21817.869} C_VEL
LIN {X 0,Y 220.049,Z 490.159,A -85,B 0,C 180,E1 -21819.96,E2 -21819.96} C_VEL
LIN {X 0,Y 215.584,Z 499.283,A -85,B 0,C 180,E1 -21822.13,E2 -21822.13} C_VEL
LIN {X 0,Y 210.996,Z 507.977,A -85,B 0,C 180,E1 -21824.732,E2 -21824.732} C_VEL
LIN {X 0,Y 206.337,Z 515.932,A -85,B 0,C 180,E1 -21827.726,E2 -21827.726} C_VEL
LIN {X 0,Y 201.883,Z 523.044,A -85,B 0,C 180,E1 -21831.2,E2 -21831.2} C_VEL
LIN {X 0,Y 198.467,Z 528.206,A -85,B 0,C 180,E1 -21834.528,E2 -21834.528} C_VEL
LIN {X 0,Y 195.182,Z 532.808,A -85,B 0,C 180,E1 -21838.527,E2 -21838.527} C_VEL
LIN {X 0,Y 193.239,Z 535.387,A -85,B 0,C 180,E1 -21841.785,E2 -21841.785} C_VEL
LIN {X 0,Y 191.373,Z 537.549,A -85,B 0,C 180,E1 -21846.175,E2 -21846.175} C_VEL
LIN {X 0,Y 190.265,Z 538.275,A -85,B 0,C 180,E1 -21850.584,E2 -21850.584} C_VEL
LIN {X 0,Y 189.898,Z 537.579,A -85,B 0,C 180,E1 -21854.986,E2 -21854.986} C_VEL
LIN {X 0,Y 189.92,Z 535.48,A -85,B 0,C 180,E1 -21859.338,E2 -21859.338} C_VEL
LIN {X 0,Y 190.526,Z 531.962,A -85,B 0,C 180,E1 -21863.647,E2 -21863.647} C_VEL
LIN {X 0,Y 191.237,Z 528.387,A -85,B 0,C 180,E1 -21866.84,E2 -21866.84} C_VEL
LIN {X 0,Y 192.252,Z 523.847,A -85,B 0,C 180,E1 -21870,E2 -21870} C_VEL
LIN {X 0,Y 193.935,Z 517.313,A -85,B 0,C 180,E1 -21873.636,E2 -21873.636} C_VEL
LIN {X 0,Y 196.308,Z 509.203,A -85,B 0,C 180,E1 -21877.198,E2 -21877.198} C_VEL
LIN {X 0,Y 198.846,Z 500.709,A -85,B 0,C 180,E1 -21880.179,E2 -21880.179} C_VEL
LIN {X 0,Y 201.648,Z 491.107,A -85,B 0,C 180,E1 -21882.914,E2 -21882.914} C_VEL
LIN {X 0,Y 204.773,Z 479.83,A -85,B 0,C 180,E1 -21885.485,E2 -21885.485} C_VEL
LIN {X 0,Y 207.717,Z 467.504,A -85,B 0,C 180,E1 -21887.729,E2 -21887.729} C_VEL
LIN {X 0,Y 209.928,Z 456.769,A -85,B 0,C 180,E1 -21889.305,E2 -21889.305} C_VEL
LIN {X 0,Y 212.293,Z 444.329,A -85,B 0,C 180,E1 -21890.72,E2 -21890.72} C_VEL
LIN {X 0,Y 214.193,Z 430.587,A -85,B 0,C 180,E1 -21891.915,E2 -21891.915} C_VEL
LIN {X 0,Y 215.653,Z 416.277,A -85,B 0,C 180,E1 -21892.768,E2 -21892.768} C_VEL
LIN {X 0,Y 216.783,Z 396.358,A -85,B 0,C 180,E1 -21893.472,E2 -21893.472} C_VEL
LIN {X 0,Y 219.845,Z 336.292,A -85,B 0,C 180,E1 -21895.289,E2 -21895.289} C_VEL
LIN {X 0,Y 213.948,Z 321.199,A -85,B 0,C 180,E1 -21896.972,E2 -21896.972} C_VEL
LIN {X 0,Y 205.525,Z 305.418,A -85,B 0,C 180,E1 -21899.36,E2 -21899.36} C_VEL
LIN {X 0,Y 197.602,Z 292.618,A -85,B 0,C 180,E1 -21901.767,E2 -21901.767} C_VEL
LIN {X 0,Y 195.419,Z 289.137,A -85,B 0,C 180,E1 -21902.476,E2 -21902.476} C_VEL
LIN {X 0,Y 193.166,Z 286.178,A -85,B 0,C 180,E1 -21903.201,E2 -21903.201} C_VEL
LIN {X 0,Y 192.588,Z 284.117,A -85,B 0,C 180,E1 -21903.5,E2 -21903.5} C_VEL
LIN {X 0,Y 192.591,Z 284.119,A -85,B 0,C 180,E1 -21908.342,E2 -21908.342} C_VEL
LIN {X 0,Y 192.612,Z 284.117,A -85,B 0,C 180,E1 -21913.139,E2 -21913.139} C_VEL
LIN {X 0,Y 192.619,Z 284.095,A -85,B 0,C 180,E1 -21916.863,E2 -21916.863} C_VEL
LIN {X 0,Y 192.605,Z 284.111,A -85,B 0,C 180,E1 -21921.665,E2 -21921.665} C_VEL
LIN {X 0,Y 192.593,Z 284.11,A -85,B 0,C 180,E1 -21926.817,E2 -21926.817} C_VEL
LIN {X 0,Y 192.658,Z 284.088,A -85,B 0,C 180,E1 -21931.694,E2 -21931.694} C_VEL
LIN {X 0,Y 192.699,Z 284.101,A -85,B 0,C 180,E1 -21936.351,E2 -21936.351} C_VEL
LIN {X 0,Y 192.726,Z 284.1,A -85,B 0,C 180,E1 -21941.46,E2 -21941.46} C_VEL
LIN {X 0,Y 192.759,Z 284.091,A -85,B 0,C 180,E1 -21945.216,E2 -21945.216} C_VEL
LIN {X 0,Y 192.941,Z 284.072,A -85,B 0,C 180,E1 -21949.569,E2 -21949.569} C_VEL
LIN {X 0,Y 192.981,Z 284.041,A -85,B 0,C 180,E1 -21953.731,E2 -21953.731} C_VEL
LIN {X 0,Y 193.259,Z 284.036,A -85,B 0,C 180,E1 -21957.919,E2 -21957.919} C_VEL
LIN {X 0,Y 193.44,Z 284.006,A -85,B 0,C 180,E1 -21960.003,E2 -21960.003} C_VEL
LIN {X 0,Y 192.968,Z 284.047,A -85,B 0,C 180,E1 -21964.18,E2 -21964.18} C_VEL
LIN {X 0,Y 193.035,Z 284.064,A -85,B 0,C 180,E1 -21968.377,E2 -21968.377} C_VEL
LIN {X 0,Y 192.8,Z 284.066,A -85,B 0,C 180,E1 -21972.636,E2 -21972.636} C_VEL
LIN {X 0,Y 192.756,Z 284.099,A -85,B 0,C 180,E1 -21976.962,E2 -21976.962} C_VEL
LIN {X 0,Y 192.616,Z 284.117,A -85,B 0,C 180,E1 -21981.402,E2 -21981.402} C_VEL
LIN {X 0,Y 192.648,Z 284.109,A -85,B 0,C 180,E1 -21984.216,E2 -21984.216} C_VEL
LIN {X 0,Y 192.651,Z 284.113,A -85,B 0,C 180,E1 -21988.894,E2 -21988.894} C_VEL
LIN {X 0,Y 192.599,Z 284.121,A -85,B 0,C 180,E1 -21993.189,E2 -21993.189} C_VEL
LIN {X 0,Y 192.555,Z 284.124,A -85,B 0,C 180,E1 -21998.354,E2 -21998.354} C_VEL
LIN {X 0,Y 192.542,Z 284.128,A -85,B 0,C 180,E1 -22001.773,E2 -22001.773} C_VEL
LIN {X 0,Y 192.728,Z 285.079,A -85,B 0,C 180,E1 -22002.251,E2 -22002.251} C_VEL
LIN {X 0,Y 194.031,Z 287.66,A -85,B 0,C 180,E1 -22002.721,E2 -22002.721} C_VEL
LIN {X 0,Y 196.301,Z 291.264,A -85,B 0,C 180,E1 -22003.474,E2 -22003.474} C_VEL
LIN {X 0,Y 201.422,Z 300.704,A -85,B 0,C 180,E1 -22005.142,E2 -22005.142} C_VEL
LIN {X 0,Y 208.181,Z 314.262,A -85,B 0,C 180,E1 -22007.212,E2 -22007.212} C_VEL
LIN {X 0,Y 214.619,Z 329.865,A -85,B 0,C 180,E1 -22009.131,E2 -22009.131} C_VEL
LIN {X 0,Y 217.517,Z 337.701,A -85,B 0,C 180,E1 -22009.979,E2 -22009.979} C_VEL
LIN {X 0,Y 218.448,Z 341.198,A -85,B 0,C 180,E1 -22010.284,E2 -22010.284} C_VEL
LIN {X 0,Y 218.465,Z 344.999,A -85,B 0,C 180,E1 -22010.436,E2 -22010.436} C_VEL
LIN {X 0,Y 217.349,Z 350.849,A -85,B 0,C 180,E1 -22010.469,E2 -22010.469} C_VEL
LIN {X 0,Y 214.131,Z 360.841,A -85,B 0,C 180,E1 -22010.292,E2 -22010.292} C_VEL
LIN {X 0,Y 212.725,Z 367.004,A -85,B 0,C 180,E1 -22010.287,E2 -22010.287} C_VEL
LIN {X 0,Y 212.529,Z 369.092,A -85,B 0,C 180,E1 -22010.336,E2 -22010.336} C_VEL
LIN {X 0,Y 209.706,Z 423.114,A -85,B 0,C 180,E1 -22012.066,E2 -22012.066} C_VEL
LIN {X 0,Y 208.294,Z 437.217,A -85,B 0,C 180,E1 -22012.831,E2 -22012.831} C_VEL
LIN {X 0,Y 206.057,Z 451.495,A -85,B 0,C 180,E1 -22013.961,E2 -22013.961} C_VEL
LIN {X 0,Y 203.234,Z 465.598,A -85,B 0,C 180,E1 -22015.511,E2 -22015.511} C_VEL
LIN {X 0,Y 200.456,Z 478.086,A -85,B 0,C 180,E1 -22017.349,E2 -22017.349} C_VEL
LIN {X 0,Y 198.055,Z 487.382,A -85,B 0,C 180,E1 -22019.034,E2 -22019.034} C_VEL
LIN {X 0,Y 195.043,Z 498.364,A -85,B 0,C 180,E1 -22021.482,E2 -22021.482} C_VEL
LIN {X 0,Y 192.197,Z 507.523,A -85,B 0,C 180,E1 -22023.973,E2 -22023.973} C_VEL
LIN {X 0,Y 189.41,Z 516.722,A -85,B 0,C 180,E1 -22027.071,E2 -22027.071} C_VEL
LIN {X 0,Y 186.893,Z 525.504,A -85,B 0,C 180,E1 -22030.79,E2 -22030.79} C_VEL
LIN {X 0,Y 185.076,Z 532.569,A -85,B 0,C 180,E1 -22034.585,E2 -22034.585} C_VEL
LIN {X 0,Y 183.94,Z 537.434,A -85,B 0,C 180,E1 -22037.869,E2 -22037.869} C_VEL
LIN {X 0,Y 183.278,Z 542.448,A -85,B 0,C 180,E1 -22042.287,E2 -22042.287} C_VEL
LIN {X 0,Y 183.06,Z 545.837,A -85,B 0,C 180,E1 -22046.586,E2 -22046.586} C_VEL
LIN {X 0,Y 183.205,Z 547.552,A -85,B 0,C 180,E1 -22050,E2 -22050} C_VEL
LIN {X 0,Y 183.039,Z 548.529,A -85,B 0,C 180,E1 -22054.404,E2 -22054.404} C_VEL
LIN {X 0,Y 183.411,Z 548.188,A -85,B 0,C 180,E1 -22058.816,E2 -22058.816} C_VEL
LIN {X 0,Y 184.505,Z 546.543,A -85,B 0,C 180,E1 -22063.211,E2 -22063.211} C_VEL
LIN {X 0,Y 186.62,Z 543.569,A -85,B 0,C 180,E1 -22067.534,E2 -22067.534} C_VEL
LIN {X 0,Y 189.59,Z 539.185,A -85,B 0,C 180,E1 -22071.758,E2 -22071.758} C_VEL
LIN {X 0,Y 193.606,Z 533.271,A -85,B 0,C 180,E1 -22075.823,E2 -22075.823} C_VEL
LIN {X 0,Y 197.941,Z 526.652,A -85,B 0,C 180,E1 -22079.221,E2 -22079.221} C_VEL
LIN {X 0,Y 203.01,Z 518.46,A -85,B 0,C 180,E1 -22082.451,E2 -22082.451} C_VEL
LIN {X 0,Y 207.904,Z 509.943,A -85,B 0,C 180,E1 -22085.075,E2 -22085.075} C_VEL
LIN {X 0,Y 213.224,Z 499.36,A -85,B 0,C 180,E1 -22087.67,E2 -22087.67} C_VEL
LIN {X 0,Y 217.816,Z 489.393,A -85,B 0,C 180,E1 -22089.586,E2 -22089.586} C_VEL
LIN {X 0,Y 222.369,Z 478.25,A -85,B 0,C 180,E1 -22091.28,E2 -22091.28} C_VEL
LIN {X 0,Y 226.529,Z 466.144,A -85,B 0,C 180,E1 -22092.738,E2 -22092.738} C_VEL
LIN {X 0,Y 230.391,Z 452.707,A -85,B 0,C 180,E1 -22093.944,E2 -22093.944} C_VEL
LIN {X 0,Y 233.464,Z 438.697,A -85,B 0,C 180,E1 -22094.872,E2 -22094.872} C_VEL
LIN {X 0,Y 235.728,Z 423.927,A -85,B 0,C 180,E1 -22095.533,E2 -22095.533} C_VEL
LIN {X 0,Y 238.493,Z 387.133,A -85,B 0,C 180,E1 -22096.574,E2 -22096.574} C_VEL
LIN {X 0,Y 239.854,Z 366.673,A -85,B 0,C 180,E1 -22097.151,E2 -22097.151} C_VEL
LIN {X 0,Y 234.907,Z 355.132,A -85,B 0,C 180,E1 -22099.374,E2 -22099.374} C_VEL
LIN {X 0,Y 229.619,Z 344.377,A -85,B 0,C 180,E1 -22101.945,E2 -22101.945} C_VEL
LIN {X 0,Y 224.285,Z 334.825,A -85,B 0,C 180,E1 -22104.794,E2 -22104.794} C_VEL
LIN {X 0,Y 221.576,Z 330.248,A -85,B 0,C 180,E1 -22106.381,E2 -22106.381} C_VEL
LIN {X 0,Y 217.655,Z 323.957,A -85,B 0,C 180,E1 -22108.891,E2 -22108.891} C_VEL
LIN {X 0,Y 215.281,Z 320.299,A -85,B 0,C 180,E1 -22110.589,E2 -22110.589} C_VEL
LIN {X 0,Y 212.038,Z 315.406,A -85,B 0,C 180,E1 -22113.192,E2 -22113.192} C_VEL
LIN {X 0,Y 207.382,Z 308.813,A -85,B 0,C 180,E1 -22117.748,E2 -22117.748} C_VEL
LIN {X 0,Y 204.57,Z 306.373,A -85,B 0,C 180,E1 -22121.176,E2 -22121.176} C_VEL
LIN {X 0,Y 203.088,Z 303.209,A -85,B 0,C 180,E1 -22123.925,E2 -22123.925} C_VEL
LIN {X 0,Y 200.589,Z 301.62,A -85,B 0,C 180,E1 -22131.941,E2 -22131.941} C_VEL
LIN {X 0,Y 201.728,Z 302.215,A -85,B 0,C 180,E1 -22139.498,E2 -22139.498} C_VEL
LIN {X 0,Y 203.472,Z 303.451,A -85,B 0,C 180,E1 -22143.174,E2 -22143.174} C_VEL
LIN {X 0,Y 204.859,Z 306.276,A -85,B 0,C 180,E1 -22145.599,E2 -22145.599} C_VEL
LIN {X 0,Y 207.822,Z 309.001,A -85,B 0,C 180,E1 -22149.118,E2 -22149.118} C_VEL
LIN {X 0,Y 210.053,Z 312.544,A -85,B 0,C 180,E1 -22151.441,E2 -22151.441} C_VEL
LIN {X 0,Y 212.029,Z 314.483,A -85,B 0,C 180,E1 -22153.139,E2 -22153.139} C_VEL
LIN {X 0,Y 214.688,Z 318.164,A -85,B 0,C 180,E1 -22155.281,E2 -22155.281} C_VEL
LIN {X 0,Y 216.094,Z 320.01,A -85,B 0,C 180,E1 -22156.313,E2 -22156.313} C_VEL
LIN {X 0,Y 219.529,Z 324.654,A -85,B 0,C 180,E1 -22158.608,E2 -22158.608} C_VEL
LIN {X 0,Y 222.939,Z 329.385,A -85,B 0,C 180,E1 -22160.648,E2 -22160.648} C_VEL
LIN {X 0,Y 227.675,Z 336.347,A -85,B 0,C 180,E1 -22163.21,E2 -22163.21} C_VEL
LIN {X 0,Y 232.31,Z 343.831,A -85,B 0,C 180,E1 -22165.491,E2 -22165.491} C_VEL
LIN {X 0,Y 237.437,Z 353.815,A -85,B 0,C 180,E1 -22167.849,E2 -22167.849} C_VEL
LIN {X 0,Y 240.318,Z 359.911,A -85,B 0,C 180,E1 -22169.09,E2 -22169.09} C_VEL
LIN {X 0,Y 236.287,Z 414.84,A -85,B 0,C 180,E1 -22170.607,E2 -22170.607} C_VEL
LIN {X 0,Y 234.282,Z 428.95,A -85,B 0,C 180,E1 -22171.249,E2 -22171.249} C_VEL
LIN {X 0,Y 231.435,Z 442.792,A -85,B 0,C 180,E1 -22172.171,E2 -22172.171} C_VEL
LIN {X 0,Y 228.126,Z 455.354,A -85,B 0,C 180,E1 -22173.319,E2 -22173.319} C_VEL
LIN {X 0,Y 224.103,Z 467.862,A -85,B 0,C 180,E1 -22174.817,E2 -22174.817} C_VEL
LIN {X 0,Y 219.774,Z 479.165,A -85,B 0,C 180,E1 -22176.541,E2 -22176.541} C_VEL
LIN {X 0,Y 214.857,Z 490.184,A -85,B 0,C 180,E1 -22178.654,E2 -22178.654} C_VEL
LIN {X 0,Y 209.751,Z 500.176,A -85,B 0,C 180,E1 -22181.073,E2 -22181.073} C_VEL
LIN {X 0,Y 204.715,Z 509.192,A -85,B 0,C 180,E1 -22183.869,E2 -22183.869} C_VEL
LIN {X 0,Y 199.385,Z 517.705,A -85,B 0,C 180,E1 -22187.273,E2 -22187.273} C_VEL
LIN {X 0,Y 194.86,Z 524.462,A -85,B 0,C 180,E1 -22190.865,E2 -22190.865} C_VEL
LIN {X 0,Y 191.58,Z 529.093,A -85,B 0,C 180,E1 -22194.06,E2 -22194.06} C_VEL
LIN {X 0,Y 188.034,Z 533.677,A -85,B 0,C 180,E1 -22198.449,E2 -22198.449} C_VEL
LIN {X 0,Y 185.475,Z 536.686,A -85,B 0,C 180,E1 -22202.955,E2 -22202.955} C_VEL
LIN {X 0,Y 183.828,Z 538.222,A -85,B 0,C 180,E1 -22207.524,E2 -22207.524} C_VEL
LIN {X 0,Y 182.976,Z 538.34,A -85,B 0,C 180,E1 -22212.106,E2 -22212.106} C_VEL
LIN {X 0,Y 182.754,Z 537.065,A -85,B 0,C 180,E1 -22216.66,E2 -22216.66} C_VEL
LIN {X 0,Y 182.981,Z 534.379,A -85,B 0,C 180,E1 -22221.163,E2 -22221.163} C_VEL
LIN {X 0,Y 183.596,Z 531.52,A -85,B 0,C 180,E1 -22224.389,E2 -22224.389} C_VEL
LIN {X 0,Y 184.357,Z 527.589,A -85,B 0,C 180,E1 -22227.816,E2 -22227.816} C_VEL
LIN {X 0,Y 185.533,Z 522.871,A -85,B 0,C 180,E1 -22231.085,E2 -22231.085} C_VEL
LIN {X 0,Y 187.493,Z 516.018,A -85,B 0,C 180,E1 -22234.838,E2 -22234.838} C_VEL
LIN {X 0,Y 190.077,Z 507.516,A -85,B 0,C 180,E1 -22238.505,E2 -22238.505} C_VEL
LIN {X 0,Y 192.859,Z 498.636,A -85,B 0,C 180,E1 -22241.562,E2 -22241.562} C_VEL
LIN {X 0,Y 196.084,Z 487.885,A -85,B 0,C 180,E1 -22244.53,E2 -22244.53} C_VEL
LIN {X 0,Y 199.07,Z 477.012,A -85,B 0,C 180,E1 -22246.933,E2 -22246.933} C_VEL
LIN {X 0,Y 201.912,Z 465.137,A -85,B 0,C 180,E1 -22249.045,E2 -22249.045} C_VEL
LIN {X 0,Y 204.408,Z 453.737,A -85,B 0,C 180,E1 -22250.635,E2 -22250.635} C_VEL
LIN {X 0,Y 206.802,Z 440.434,A -85,B 0,C 180,E1 -22252.083,E2 -22252.083} C_VEL
LIN {X 0,Y 208.596,Z 426.785,A -85,B 0,C 180,E1 -22253.189,E2 -22253.189} C_VEL
LIN {X 0,Y 209.972,Z 412.031,A -85,B 0,C 180,E1 -22253.97,E2 -22253.97} C_VEL
LIN {X 0,Y 213.877,Z 338.057,A -85,B 0,C 180,E1 -22256.298,E2 -22256.298} C_VEL
LIN {X 0,Y 208.693,Z 324.722,A -85,B 0,C 180,E1 -22257.861,E2 -22257.861} C_VEL
LIN {X 0,Y 200.631,Z 309.532,A -85,B 0,C 180,E1 -22260.267,E2 -22260.267} C_VEL
LIN {X 0,Y 193.007,Z 297.123,A -85,B 0,C 180,E1 -22262.705,E2 -22262.705} C_VEL
LIN {X 0,Y 188.588,Z 290.355,A -85,B 0,C 180,E1 -22264.231,E2 -22264.231} C_VEL
LIN {X 0,Y 186.168,Z 287.115,A -85,B 0,C 180,E1 -22265.09,E2 -22265.09} C_VEL
LIN {X 0,Y 185.539,Z 284.996,A -85,B 0,C 180,E1 -22265.419,E2 -22265.419} C_VEL
LIN {X 0,Y 185.558,Z 284.98,A -85,B 0,C 180,E1 -22270.761,E2 -22270.761} C_VEL
LIN {X 0,Y 185.576,Z 284.974,A -85,B 0,C 180,E1 -22276.017,E2 -22276.017} C_VEL
LIN {X 0,Y 185.557,Z 284.994,A -85,B 0,C 180,E1 -22279.923,E2 -22279.923} C_VEL
LIN {X 0,Y 185.568,Z 284.974,A -85,B 0,C 180,E1 -22282.706,E2 -22282.706} C_VEL
LIN {X 0,Y 185.538,Z 284.996,A -85,B 0,C 180,E1 -22287.978,E2 -22287.978} C_VEL
LIN {X 0,Y 185.575,Z 284.98,A -85,B 0,C 180,E1 -22290.578,E2 -22290.578} C_VEL
LIN {X 0,Y 185.581,Z 284.977,A -85,B 0,C 180,E1 -22295.385,E2 -22295.385} C_VEL
LIN {X 0,Y 185.601,Z 284.984,A -85,B 0,C 180,E1 -22300.078,E2 -22300.078} C_VEL
LIN {X 0,Y 185.69,Z 284.973,A -85,B 0,C 180,E1 -22304.64,E2 -22304.64} C_VEL
LIN {X 0,Y 185.884,Z 284.951,A -85,B 0,C 180,E1 -22309.421,E2 -22309.421} C_VEL
LIN {X 0,Y 185.943,Z 284.915,A -85,B 0,C 180,E1 -22313.492,E2 -22313.492} C_VEL
LIN {X 0,Y 186.203,Z 284.914,A -85,B 0,C 180,E1 -22317.84,E2 -22317.84} C_VEL
LIN {X 0,Y 186.403,Z 284.882,A -85,B 0,C 180,E1 -22320.003,E2 -22320.003} C_VEL
LIN {X 0,Y 185.915,Z 284.925,A -85,B 0,C 180,E1 -22324.339,E2 -22324.339} C_VEL
LIN {X 0,Y 185.981,Z 284.941,A -85,B 0,C 180,E1 -22328.697,E2 -22328.697} C_VEL
LIN {X 0,Y 185.727,Z 284.947,A -85,B 0,C 180,E1 -22333.126,E2 -22333.126} C_VEL
LIN {X 0,Y 185.689,Z 284.98,A -85,B 0,C 180,E1 -22337.628,E2 -22337.628} C_VEL
LIN {X 0,Y 185.578,Z 284.991,A -85,B 0,C 180,E1 -22342.256,E2 -22342.256} C_VEL
LIN {X 0,Y 185.562,Z 284.991,A -85,B 0,C 180,E1 -22347.035,E2 -22347.035} C_VEL
LIN {X 0,Y 185.581,Z 284.995,A -85,B 0,C 180,E1 -22349.496,E2 -22349.496} C_VEL
LIN {X 0,Y 185.502,Z 284.999,A -85,B 0,C 180,E1 -22354.635,E2 -22354.635} C_VEL
LIN {X 0,Y 185.509,Z 285,A -85,B 0,C 180,E1 -22357.315,E2 -22357.315} C_VEL
LIN {X 0,Y 185.472,Z 285.004,A -85,B 0,C 180,E1 -22360.216,E2 -22360.216} C_VEL
LIN {X 0,Y 186.351,Z 287.622,A -85,B 0,C 180,E1 -22360.616,E2 -22360.616} C_VEL
LIN {X 0,Y 188.553,Z 290.422,A -85,B 0,C 180,E1 -22361.385,E2 -22361.385} C_VEL
LIN {X 0,Y 192.274,Z 296.648,A -85,B 0,C 180,E1 -22362.703,E2 -22362.703} C_VEL
LIN {X 0,Y 198.772,Z 308.965,A -85,B 0,C 180,E1 -22364.905,E2 -22364.905} C_VEL
LIN {X 0,Y 204.769,Z 321.851,A -85,B 0,C 180,E1 -22366.825,E2 -22366.825} C_VEL
LIN {X 0,Y 210.393,Z 336.271,A -85,B 0,C 180,E1 -22368.586,E2 -22368.586} C_VEL
LIN {X 0,Y 212.815,Z 343.188,A -85,B 0,C 180,E1 -22369.335,E2 -22369.335} C_VEL
LIN {X 0,Y 213.488,Z 350.401,A -85,B 0,C 180,E1 -22369.754,E2 -22369.754} C_VEL
LIN {X 0,Y 212.529,Z 369.092,A -85,B 0,C 180,E1 -22370.336,E2 -22370.336} C_VEL
LIN {X 0,Y 211.68,Z 374.932,A -85,B 0,C 180,E1 -22370.418,E2 -22370.418} C_VEL
LIN {X 0,Y 205.905,Z 393.888,A -85,B 0,C 180,E1 -22370.133,E2 -22370.133} C_VEL
LIN {X 0,Y 205.055,Z 399.727,A -85,B 0,C 180,E1 -22370.218,E2 -22370.218} C_VEL
LIN {X 0,Y 203.634,Z 424.4,A -85,B 0,C 180,E1 -22371.072,E2 -22371.072} C_VEL
LIN {X 0,Y 202.058,Z 438.431,A -85,B 0,C 180,E1 -22371.875,E2 -22371.875} C_VEL
LIN {X 0,Y 199.883,Z 451.783,A -85,B 0,C 180,E1 -22372.979,E2 -22372.979} C_VEL
LIN {X 0,Y 196.967,Z 465.781,A -85,B 0,C 180,E1 -22374.563,E2 -22374.563} C_VEL
LIN {X 0,Y 194.099,Z 478.166,A -85,B 0,C 180,E1 -22376.443,E2 -22376.443} C_VEL
